   1:  PR[GP1:91,1] = PR[GP1:90,1] + -18.731;
   1:  PR[GP1:91,2] = PR[GP1:90,2] + 32.374;
   1:L PR[91] 10mm/sec CNT100;
   1:  PR[GP1:91,1] = PR[GP1:90,1] + -20.880;
   1:  PR[GP1:91,2] = PR[GP1:90,2] + 33.052;
   1:L PR[91] 10mm/sec CNT100;
   1:  PR[GP1:91,1] = PR[GP1:90,1] + -27.675;
   1:  PR[GP1:91,2] = PR[GP1:90,2] + 35.074;
   1:L PR[91] 10mm/sec CNT100;
   1:  PR[GP1:91,1] = PR[GP1:90,1] + -31.879;
   1:  PR[GP1:91,2] = PR[GP1:90,2] + 35.433;
   1:L PR[91] 10mm/sec CNT100;
   1:  PR[GP1:91,1] = PR[GP1:90,1] + -39.590;
   1:  PR[GP1:91,2] = PR[GP1:90,2] + 35.208;
   1:L PR[91] 10mm/sec CNT100;
   1:  PR[GP1:91,1] = PR[GP1:90,1] + -42.034;
   1:  PR[GP1:91,2] = PR[GP1:90,2] + 34.900;
   1:L PR[91] 10mm/sec CNT100;
   1:  PR[GP1:91,1] = PR[GP1:90,1] + -53.582;
   1:  PR[GP1:91,2] = PR[GP1:90,2] + 30.630;
   1:L PR[91] 10mm/sec CNT100;
   1:  PR[GP1:91,1] = PR[GP1:90,1] + -53.589;
   1:  PR[GP1:91,2] = PR[GP1:90,2] + 30.626;
   1:L PR[91] 10mm/sec CNT100;
   1:  PR[GP1:91,1] = PR[GP1:90,1] + -63.016;
   1:  PR[GP1:91,2] = PR[GP1:90,2] + 22.850;
   1:L PR[91] 10mm/sec CNT100;
   1:  PR[GP1:91,1] = PR[GP1:90,1] + -64.107;
   1:  PR[GP1:91,2] = PR[GP1:90,2] + 21.068;
   1:L PR[91] 10mm/sec CNT100;
   1:  PR[GP1:91,1] = PR[GP1:90,1] + -69.252;
   1:  PR[GP1:91,2] = PR[GP1:90,2] + 12.300;
   1:L PR[91] 10mm/sec CNT100;
   1:  PR[GP1:91,1] = PR[GP1:90,1] + -69.934;
   1:  PR[GP1:91,2] = PR[GP1:90,2] + 8.701;
   1:L PR[91] 10mm/sec CNT100;
   1:  PR[GP1:91,1] = PR[GP1:90,1] + -71.444;
   1:  PR[GP1:91,2] = PR[GP1:90,2] + 0.282;
   1:L PR[91] 10mm/sec CNT100;
   1:  PR[GP1:91,1] = PR[GP1:90,1] + -70.746;
   1:  PR[GP1:91,2] = PR[GP1:90,2] + -3.377;
   1:L PR[91] 10mm/sec CNT100;
   1:  PR[GP1:91,1] = PR[GP1:90,1] + -69.251;
   1:  PR[GP1:91,2] = PR[GP1:90,2] + -11.744;
   1:L PR[91] 10mm/sec CNT100;
   1:  PR[GP1:91,1] = PR[GP1:90,1] + -64.107;
   1:  PR[GP1:91,2] = PR[GP1:90,2] + -20.510;
   1:L PR[91] 10mm/sec CNT100;
   1:  PR[GP1:91,1] = PR[GP1:90,1] + -63.016;
   1:  PR[GP1:91,2] = PR[GP1:90,2] + -22.292;
   1:L PR[91] 10mm/sec CNT100;
   1:  PR[GP1:91,1] = PR[GP1:90,1] + -53.589;
   1:  PR[GP1:91,2] = PR[GP1:90,2] + -30.068;
   1:L PR[91] 10mm/sec CNT100;
   1:  PR[GP1:91,1] = PR[GP1:90,1] + -53.582;
   1:  PR[GP1:91,2] = PR[GP1:90,2] + -30.072;
   1:L PR[91] 10mm/sec CNT100;
   1:  PR[GP1:91,1] = PR[GP1:90,1] + -42.034;
   1:  PR[GP1:91,2] = PR[GP1:90,2] + -34.342;
   1:L PR[91] 10mm/sec CNT100;
   1:  PR[GP1:91,1] = PR[GP1:90,1] + -39.590;
   1:  PR[GP1:91,2] = PR[GP1:90,2] + -34.650;
   1:L PR[91] 10mm/sec CNT100;
   1:  PR[GP1:91,1] = PR[GP1:90,1] + -31.879;
   1:  PR[GP1:91,2] = PR[GP1:90,2] + -34.875;
   1:L PR[91] 10mm/sec CNT100;
   1:  PR[GP1:91,1] = PR[GP1:90,1] + -27.681;
   1:  PR[GP1:91,2] = PR[GP1:90,2] + -34.516;
   1:L PR[91] 10mm/sec CNT100;
   1:  PR[GP1:91,1] = PR[GP1:90,1] + -23.858;
   1:  PR[GP1:91,2] = PR[GP1:90,2] + -33.291;
   1:L PR[91] 10mm/sec CNT100;
   1:  PR[GP1:91,1] = PR[GP1:90,1] + -18.724;
   1:  PR[GP1:91,2] = PR[GP1:90,2] + -31.812;
   1:L PR[91] 10mm/sec CNT100;
   1:  PR[GP1:91,1] = PR[GP1:90,1] + -14.436;
   1:  PR[GP1:91,2] = PR[GP1:90,2] + -29.375;
   1:L PR[91] 10mm/sec CNT100;
   1:  PR[GP1:91,1] = PR[GP1:90,1] + -11.858;
   1:  PR[GP1:91,2] = PR[GP1:90,2] + -27.972;
   1:L PR[91] 10mm/sec CNT100;
   1:  PR[GP1:91,1] = PR[GP1:90,1] + -5.874;
   1:  PR[GP1:91,2] = PR[GP1:90,2] + -22.708;
   1:L PR[91] 10mm/sec CNT100;
   1:  PR[GP1:91,1] = PR[GP1:90,1] + -5.197;
   1:  PR[GP1:91,2] = PR[GP1:90,2] + -21.887;
   1:L PR[91] 10mm/sec CNT100;
   1:  PR[GP1:91,1] = PR[GP1:90,1] + -1.808;
   1:  PR[GP1:91,2] = PR[GP1:90,2] + -17.107;
   1:L PR[91] 10mm/sec CNT100;
   1:  PR[GP1:91,1] = PR[GP1:90,1] + 1.289;
   1:L PR[91] 10mm/sec CNT100;
   1:  PR[GP1:91,1] = PR[GP1:90,1] + 4.280;
   1:  PR[GP1:91,2] = PR[GP1:90,2] + -21.758;
   1:  PR[GP1:91,3] = PR[GP1:90,3] + 40.565;
   1:L PR[91] 10mm/sec CNT100;
   1:  PR[GP1:91,1] = PR[GP1:90,1] + 5.162;
   1:  PR[GP1:91,2] = PR[GP1:90,2] + -22.831;
   1:L PR[91] 10mm/sec CNT100;
   1:  PR[GP1:91,1] = PR[GP1:90,1] + 11.120;
   1:  PR[GP1:91,2] = PR[GP1:90,2] + -28.070;
   1:L PR[91] 10mm/sec CNT100;
   1:  PR[GP1:91,1] = PR[GP1:90,1] + 16.147;
   1:  PR[GP1:91,2] = PR[GP1:90,2] + -30.798;
   1:L PR[91] 10mm/sec CNT100;
   1:  PR[GP1:91,1] = PR[GP1:90,1] + 18.170;
   1:  PR[GP1:91,2] = PR[GP1:90,2] + -31.944;
   1:L PR[91] 10mm/sec CNT100;
   1:  PR[GP1:91,1] = PR[GP1:90,1] + 19.162;
   1:  PR[GP1:91,2] = PR[GP1:90,2] + -32.258;
   1:L PR[91] 10mm/sec CNT100;
   1:  PR[GP1:91,1] = PR[GP1:90,1] + 26.811;
   1:  PR[GP1:91,2] = PR[GP1:90,2] + -34.534;
   1:L PR[91] 10mm/sec CNT100;
   1:  PR[GP1:91,1] = PR[GP1:90,1] + 31.532;
   1:  PR[GP1:91,2] = PR[GP1:90,2] + -34.940;
   1:L PR[91] 10mm/sec CNT100;
   1:  PR[GP1:91,1] = PR[GP1:90,1] + 38.345;
   1:  PR[GP1:91,2] = PR[GP1:90,2] + -34.741;
   1:L PR[91] 10mm/sec CNT100;
   1:  PR[GP1:91,1] = PR[GP1:90,1] + 41.413;
   1:  PR[GP1:91,2] = PR[GP1:90,2] + -34.357;
   1:L PR[91] 10mm/sec CNT100;
   1:  PR[GP1:91,1] = PR[GP1:90,1] + 52.707;
   1:  PR[GP1:91,2] = PR[GP1:90,2] + -30.191;
   1:L PR[91] 10mm/sec CNT100;
   1:  PR[GP1:91,1] = PR[GP1:90,1] + 53.122;
   1:  PR[GP1:91,2] = PR[GP1:90,2] + -29.937;
   1:L PR[91] 10mm/sec CNT100;
   1:  PR[GP1:91,1] = PR[GP1:90,1] + 62.401;
   1:  PR[GP1:91,2] = PR[GP1:90,2] + -22.260;
   1:L PR[91] 10mm/sec CNT100;
   1:  PR[GP1:91,1] = PR[GP1:90,1] + 63.095;
   1:  PR[GP1:91,2] = PR[GP1:90,2] + -21.128;
   1:L PR[91] 10mm/sec CNT100;
   1:  PR[GP1:91,1] = PR[GP1:90,1] + 68.617;
   1:  PR[GP1:91,2] = PR[GP1:90,2] + -11.744;
   1:L PR[91] 10mm/sec CNT100;
   1:  PR[GP1:91,1] = PR[GP1:90,1] + 69.156;
   1:  PR[GP1:91,2] = PR[GP1:90,2] + -8.896;
   1:L PR[91] 10mm/sec CNT100;
   1:  PR[GP1:91,1] = PR[GP1:90,1] + 70.798;
   1:  PR[GP1:91,2] = PR[GP1:90,2] + 0.276;
   1:L PR[91] 10mm/sec CNT100;
   1:  PR[GP1:91,1] = PR[GP1:90,1] + 70.220;
   1:  PR[GP1:91,2] = PR[GP1:90,2] + 3.310;
   1:L PR[91] 10mm/sec CNT100;
   1:  PR[GP1:91,1] = PR[GP1:90,1] + 68.615;
   1:  PR[GP1:91,2] = PR[GP1:90,2] + 12.305;
   1:L PR[91] 10mm/sec CNT100;
   1:  PR[GP1:91,1] = PR[GP1:90,1] + 63.095;
   1:  PR[GP1:91,2] = PR[GP1:90,2] + 21.686;
   1:L PR[91] 10mm/sec CNT100;
   1:  PR[GP1:91,1] = PR[GP1:90,1] + 62.401;
   1:  PR[GP1:91,2] = PR[GP1:90,2] + 22.818;
   1:L PR[91] 10mm/sec CNT100;
   1:  PR[GP1:91,1] = PR[GP1:90,1] + 53.122;
   1:  PR[GP1:91,2] = PR[GP1:90,2] + 30.495;
   1:L PR[91] 10mm/sec CNT100;
   1:  PR[GP1:91,1] = PR[GP1:90,1] + 52.707;
   1:  PR[GP1:91,2] = PR[GP1:90,2] + 30.749;
   1:L PR[91] 10mm/sec CNT100;
   1:  PR[GP1:91,1] = PR[GP1:90,1] + 43.327;
   1:  PR[GP1:91,2] = PR[GP1:90,2] + 34.223;
   1:L PR[91] 10mm/sec CNT100;
   1:  PR[GP1:91,1] = PR[GP1:90,1] + 41.415;
   1:  PR[GP1:91,2] = PR[GP1:90,2] + 34.915;
   1:L PR[91] 10mm/sec CNT100;
   1:  PR[GP1:91,1] = PR[GP1:90,1] + 38.345;
   1:  PR[GP1:91,2] = PR[GP1:90,2] + 35.299;
   1:L PR[91] 10mm/sec CNT100;
   1:  PR[GP1:91,1] = PR[GP1:90,1] + 31.532;
   1:  PR[GP1:91,2] = PR[GP1:90,2] + 35.498;
   1:L PR[91] 10mm/sec CNT100;
   1:  PR[GP1:91,1] = PR[GP1:90,1] + 26.818;
   1:  PR[GP1:91,2] = PR[GP1:90,2] + 35.093;
   1:L PR[91] 10mm/sec CNT100;
   1:  PR[GP1:91,1] = PR[GP1:90,1] + 23.739;
   1:  PR[GP1:91,2] = PR[GP1:90,2] + 34.106;
   1:L PR[91] 10mm/sec CNT100;
   1:  PR[GP1:91,1] = PR[GP1:90,1] + 18.163;
   1:  PR[GP1:91,2] = PR[GP1:90,2] + 32.499;
   1:L PR[91] 10mm/sec CNT100;
   1:  PR[GP1:91,1] = PR[GP1:90,1] + 16.146;
   1:  PR[GP1:91,2] = PR[GP1:90,2] + 31.356;
   1:L PR[91] 10mm/sec CNT100;
   1:  PR[GP1:91,1] = PR[GP1:90,1] + 11.256;
   1:  PR[GP1:91,2] = PR[GP1:90,2] + 28.716;
   1:L PR[91] 10mm/sec CNT100;
   1:  PR[GP1:91,1] = PR[GP1:90,1] + 10.671;
   1:  PR[GP1:91,2] = PR[GP1:90,2] + 28.240;
   1:L PR[91] 10mm/sec CNT100;
   1:  PR[GP1:91,1] = PR[GP1:90,1] + 5.156;
   1:  PR[GP1:91,2] = PR[GP1:90,2] + 23.383;
   1:L PR[91] 10mm/sec CNT100;
   1:  PR[GP1:91,1] = PR[GP1:90,1] + 4.259;
   1:  PR[GP1:91,2] = PR[GP1:90,2] + 22.289;
   1:L PR[91] 10mm/sec CNT100;
   1:  PR[GP1:91,1] = PR[GP1:90,1] + 1.201;
   1:  PR[GP1:91,2] = PR[GP1:90,2] + 17.990;
   1:L PR[91] 10mm/sec CNT100;
   1:  PR[GP1:91,1] = PR[GP1:90,1] + -1.721;
   1:L PR[91] 10mm/sec CNT100;
   1:  PR[GP1:91,1] = PR[GP1:90,1] + -4.761;
   1:  PR[GP1:91,2] = PR[GP1:90,2] + 22.278;
   1:L PR[91] 10mm/sec CNT100;
   1:  PR[GP1:91,1] = PR[GP1:90,1] + -5.643;
   1:  PR[GP1:91,2] = PR[GP1:90,2] + 23.348;
   1:L PR[91] 10mm/sec CNT100;
   1:  PR[GP1:91,1] = PR[GP1:90,1] + -11.163;
   1:  PR[GP1:91,2] = PR[GP1:90,2] + 28.209;
   1:L PR[91] 10mm/sec CNT100;
   1:  PR[GP1:91,1] = PR[GP1:90,1] + -11.750;
   1:  PR[GP1:91,2] = PR[GP1:90,2] + 28.687;
   1:L PR[91] 10mm/sec CNT100;
   1:  PR[GP1:91,1] = PR[GP1:90,1] + -16.673;
   1:  PR[GP1:91,2] = PR[GP1:90,2] + 31.352;
   1:L PR[91] 10mm/sec CNT100;
   1:  PR[GP1:91,1] = PR[GP1:90,1] + -18.703;
   1:  PR[GP1:91,2] = PR[GP1:90,2] + 32.506;
   1:L PR[91] 10mm/sec CNT100;
   1:  PR[GP1:91,1] = PR[GP1:90,1] + -19.698;
   1:  PR[GP1:91,2] = PR[GP1:90,2] + 32.820;
   1:L PR[91] 10mm/sec CNT100;
   1:  PR[GP1:91,1] = PR[GP1:90,1] + -27.337;
   1:  PR[GP1:91,2] = PR[GP1:90,2] + 35.093;
   1:L PR[91] 10mm/sec CNT100;
   1:  PR[GP1:91,1] = PR[GP1:90,1] + -32.070;
   1:  PR[GP1:91,2] = PR[GP1:90,2] + 35.498;
   1:L PR[91] 10mm/sec CNT100;
   1:  PR[GP1:91,1] = PR[GP1:90,1] + -38.884;
   1:  PR[GP1:91,2] = PR[GP1:90,2] + 35.298;
   1:L PR[91] 10mm/sec CNT100;
   1:  PR[GP1:91,1] = PR[GP1:90,1] + -41.955;
   1:  PR[GP1:91,2] = PR[GP1:90,2] + 34.912;
   1:L PR[91] 10mm/sec CNT100;
   1:  PR[GP1:91,1] = PR[GP1:90,1] + -53.238;
   1:  PR[GP1:91,2] = PR[GP1:90,2] + 30.743;
   1:L PR[91] 10mm/sec CNT100;
   1:  PR[GP1:91,1] = PR[GP1:90,1] + -53.655;
   1:  PR[GP1:91,2] = PR[GP1:90,2] + 30.487;
   1:L PR[91] 10mm/sec CNT100;
   1:  PR[GP1:91,1] = PR[GP1:90,1] + -62.929;
   1:  PR[GP1:91,2] = PR[GP1:90,2] + 22.824;
   1:L PR[91] 10mm/sec CNT100;
   1:  PR[GP1:91,1] = PR[GP1:90,1] + -63.623;
   1:  PR[GP1:91,2] = PR[GP1:90,2] + 21.691;
   1:L PR[91] 10mm/sec CNT100;
   1:  PR[GP1:91,1] = PR[GP1:90,1] + -69.144;
   1:  PR[GP1:91,2] = PR[GP1:90,2] + 12.283;
   1:L PR[91] 10mm/sec CNT100;
   1:  PR[GP1:91,1] = PR[GP1:90,1] + -69.683;
   1:  PR[GP1:91,2] = PR[GP1:90,2] + 9.438;
   1:L PR[91] 10mm/sec CNT100;
   1:  PR[GP1:91,1] = PR[GP1:90,1] + -71.325;
   1:  PR[GP1:91,2] = PR[GP1:90,2] + 0.282;
   1:L PR[91] 10mm/sec CNT100;
   1:  PR[GP1:91,1] = PR[GP1:90,1] + -70.746;
   1:  PR[GP1:91,2] = PR[GP1:90,2] + -2.749;
   1:L PR[91] 10mm/sec CNT100;
   1:  PR[GP1:91,1] = PR[GP1:90,1] + -69.142;
   1:  PR[GP1:91,2] = PR[GP1:90,2] + -11.727;
   1:L PR[91] 10mm/sec CNT100;
   1:  PR[GP1:91,1] = PR[GP1:90,1] + -63.623;
   1:  PR[GP1:91,2] = PR[GP1:90,2] + -21.133;
   1:L PR[91] 10mm/sec CNT100;
   1:  PR[GP1:91,1] = PR[GP1:90,1] + -62.929;
   1:  PR[GP1:91,2] = PR[GP1:90,2] + -22.266;
   1:L PR[91] 10mm/sec CNT100;
   1:  PR[GP1:91,1] = PR[GP1:90,1] + -53.655;
   1:  PR[GP1:91,2] = PR[GP1:90,2] + -29.929;
   1:L PR[91] 10mm/sec CNT100;
   1:  PR[GP1:91,1] = PR[GP1:90,1] + -53.238;
   1:  PR[GP1:91,2] = PR[GP1:90,2] + -30.185;
   1:L PR[91] 10mm/sec CNT100;
   1:  PR[GP1:91,1] = PR[GP1:90,1] + -43.863;
   1:  PR[GP1:91,2] = PR[GP1:90,2] + -33.661;
   1:L PR[91] 10mm/sec CNT100;
   1:  PR[GP1:91,1] = PR[GP1:90,1] + -41.957;
   1:  PR[GP1:91,2] = PR[GP1:90,2] + -34.354;
   1:L PR[91] 10mm/sec CNT100;
   1:  PR[GP1:91,1] = PR[GP1:90,1] + -38.884;
   1:  PR[GP1:91,2] = PR[GP1:90,2] + -34.740;
   1:L PR[91] 10mm/sec CNT100;
   1:  PR[GP1:91,1] = PR[GP1:90,1] + -32.070;
   1:  PR[GP1:91,2] = PR[GP1:90,2] + -34.940;
   1:L PR[91] 10mm/sec CNT100;
   1:  PR[GP1:91,1] = PR[GP1:90,1] + -27.344;
   1:  PR[GP1:91,2] = PR[GP1:90,2] + -34.535;
   1:L PR[91] 10mm/sec CNT100;
   1:  PR[GP1:91,1] = PR[GP1:90,1] + -24.265;
   1:  PR[GP1:91,2] = PR[GP1:90,2] + -33.549;
   1:L PR[91] 10mm/sec CNT100;
   1:  PR[GP1:91,1] = PR[GP1:90,1] + -18.697;
   1:  PR[GP1:91,2] = PR[GP1:90,2] + -31.944;
   1:L PR[91] 10mm/sec CNT100;
   1:  PR[GP1:91,1] = PR[GP1:90,1] + -16.674;
   1:  PR[GP1:91,2] = PR[GP1:90,2] + -30.794;
   1:L PR[91] 10mm/sec CNT100;
   1:  PR[GP1:91,1] = PR[GP1:90,1] + -11.614;
   1:  PR[GP1:91,2] = PR[GP1:90,2] + -28.041;
   1:L PR[91] 10mm/sec CNT100;
   1:  PR[GP1:91,1] = PR[GP1:90,1] + -5.648;
   1:  PR[GP1:91,2] = PR[GP1:90,2] + -22.797;
   1:L PR[91] 10mm/sec CNT100;
   1:  PR[GP1:91,1] = PR[GP1:90,1] + -4.767;
   1:  PR[GP1:91,2] = PR[GP1:90,2] + -21.728;
   1:L PR[91] 10mm/sec CNT100;
   1:  PR[GP1:91,1] = PR[GP1:90,1] + -1.721;
   1:  PR[GP1:91,2] = PR[GP1:90,2] + -17.432;
   1:L PR[91] 10mm/sec CNT100;
   1:  PR[GP1:91,1] = PR[GP1:90,1] + 1.203;
   1:L PR[91] 10mm/sec CNT100;
   1:  PR[GP1:91,1] = PR[GP1:90,1] + 3.847;
   1:  PR[GP1:91,2] = PR[GP1:90,2] + -21.595;
   1:  PR[GP1:91,3] = PR[GP1:90,3] + 41.175;
   1:L PR[91] 10mm/sec CNT100;
   1:  PR[GP1:91,1] = PR[GP1:90,1] + 4.935;
   1:  PR[GP1:91,2] = PR[GP1:90,2] + -22.918;
   1:L PR[91] 10mm/sec CNT100;
   1:  PR[GP1:91,1] = PR[GP1:90,1] + 10.876;
   1:  PR[GP1:91,2] = PR[GP1:90,2] + -28.138;
   1:L PR[91] 10mm/sec CNT100;
   1:  PR[GP1:91,1] = PR[GP1:90,1] + 18.113;
   1:  PR[GP1:91,2] = PR[GP1:90,2] + -32.067;
   1:L PR[91] 10mm/sec CNT100;
   1:  PR[GP1:91,1] = PR[GP1:90,1] + 26.475;
   1:  PR[GP1:91,2] = PR[GP1:90,2] + -34.553;
   1:L PR[91] 10mm/sec CNT100;
   1:  PR[GP1:91,1] = PR[GP1:90,1] + 31.723;
   1:  PR[GP1:91,2] = PR[GP1:90,2] + -35.005;
   1:L PR[91] 10mm/sec CNT100;
   1:  PR[GP1:91,1] = PR[GP1:90,1] + 37.637;
   1:  PR[GP1:91,2] = PR[GP1:90,2] + -34.832;
   1:L PR[91] 10mm/sec CNT100;
   1:  PR[GP1:91,1] = PR[GP1:90,1] + 41.332;
   1:  PR[GP1:91,2] = PR[GP1:90,2] + -34.369;
   1:L PR[91] 10mm/sec CNT100;
   1:  PR[GP1:91,1] = PR[GP1:90,1] + 52.361;
   1:  PR[GP1:91,2] = PR[GP1:90,2] + -30.305;
   1:L PR[91] 10mm/sec CNT100;
   1:  PR[GP1:91,1] = PR[GP1:90,1] + 53.185;
   1:  PR[GP1:91,2] = PR[GP1:90,2] + -29.801;
   1:L PR[91] 10mm/sec CNT100;
   1:  PR[GP1:91,1] = PR[GP1:90,1] + 62.315;
   1:  PR[GP1:91,2] = PR[GP1:90,2] + -22.234;
   1:L PR[91] 10mm/sec CNT100;
   1:  PR[GP1:91,1] = PR[GP1:90,1] + 62.611;
   1:  PR[GP1:91,2] = PR[GP1:90,2] + -21.750;
   1:L PR[91] 10mm/sec CNT100;
   1:  PR[GP1:91,1] = PR[GP1:90,1] + 68.508;
   1:  PR[GP1:91,2] = PR[GP1:90,2] + -11.728;
   1:L PR[91] 10mm/sec CNT100;
   1:  PR[GP1:91,1] = PR[GP1:90,1] + 68.904;
   1:  PR[GP1:91,2] = PR[GP1:90,2] + -9.635;
   1:L PR[91] 10mm/sec CNT100;
   1:  PR[GP1:91,1] = PR[GP1:90,1] + 70.679;
   1:  PR[GP1:91,2] = PR[GP1:90,2] + 0.276;
   1:L PR[91] 10mm/sec CNT100;
   1:  PR[GP1:91,1] = PR[GP1:90,1] + 70.220;
   1:  PR[GP1:91,2] = PR[GP1:90,2] + 2.681;
   1:L PR[91] 10mm/sec CNT100;
   1:  PR[GP1:91,1] = PR[GP1:90,1] + 68.507;
   1:  PR[GP1:91,2] = PR[GP1:90,2] + 12.289;
   1:L PR[91] 10mm/sec CNT100;
   1:  PR[GP1:91,1] = PR[GP1:90,1] + 62.611;
   1:  PR[GP1:91,2] = PR[GP1:90,2] + 22.308;
   1:L PR[91] 10mm/sec CNT100;
   1:  PR[GP1:91,1] = PR[GP1:90,1] + 62.315;
   1:  PR[GP1:91,2] = PR[GP1:90,2] + 22.792;
   1:L PR[91] 10mm/sec CNT100;
   1:  PR[GP1:91,1] = PR[GP1:90,1] + 53.185;
   1:  PR[GP1:91,2] = PR[GP1:90,2] + 30.359;
   1:L PR[91] 10mm/sec CNT100;
   1:  PR[GP1:91,1] = PR[GP1:90,1] + 52.361;
   1:  PR[GP1:91,2] = PR[GP1:90,2] + 30.863;
   1:L PR[91] 10mm/sec CNT100;
   1:  PR[GP1:91,1] = PR[GP1:90,1] + 43.637;
   1:  PR[GP1:91,2] = PR[GP1:90,2] + 34.094;
   1:L PR[91] 10mm/sec CNT100;
   1:  PR[GP1:91,1] = PR[GP1:90,1] + 41.334;
   1:  PR[GP1:91,2] = PR[GP1:90,2] + 34.927;
   1:L PR[91] 10mm/sec CNT100;
   1:  PR[GP1:91,1] = PR[GP1:90,1] + 37.637;
   1:  PR[GP1:91,2] = PR[GP1:90,2] + 35.390;
   1:L PR[91] 10mm/sec CNT100;
   1:  PR[GP1:91,1] = PR[GP1:90,1] + 31.723;
   1:  PR[GP1:91,2] = PR[GP1:90,2] + 35.563;
   1:L PR[91] 10mm/sec CNT100;
   1:  PR[GP1:91,1] = PR[GP1:90,1] + 26.481;
   1:  PR[GP1:91,2] = PR[GP1:90,2] + 35.112;
   1:L PR[91] 10mm/sec CNT100;
   1:  PR[GP1:91,1] = PR[GP1:90,1] + 24.146;
   1:  PR[GP1:91,2] = PR[GP1:90,2] + 34.364;
   1:L PR[91] 10mm/sec CNT100;
   1:  PR[GP1:91,1] = PR[GP1:90,1] + 18.110;
   1:  PR[GP1:91,2] = PR[GP1:90,2] + 32.624;
   1:L PR[91] 10mm/sec CNT100;
   1:  PR[GP1:91,1] = PR[GP1:90,1] + 11.083;
   1:  PR[GP1:91,2] = PR[GP1:90,2] + 28.830;
   1:L PR[91] 10mm/sec CNT100;
   1:  PR[GP1:91,1] = PR[GP1:90,1] + 10.186;
   1:  PR[GP1:91,2] = PR[GP1:90,2] + 28.100;
   1:L PR[91] 10mm/sec CNT100;
   1:  PR[GP1:91,1] = PR[GP1:90,1] + 4.927;
   1:  PR[GP1:91,2] = PR[GP1:90,2] + 23.469;
   1:L PR[91] 10mm/sec CNT100;
   1:  PR[GP1:91,1] = PR[GP1:90,1] + 3.822;
   1:  PR[GP1:91,2] = PR[GP1:90,2] + 22.121;
   1:L PR[91] 10mm/sec CNT100;
   1:  PR[GP1:91,1] = PR[GP1:90,1] + 1.115;
   1:  PR[GP1:91,2] = PR[GP1:90,2] + 18.315;
   1:L PR[91] 10mm/sec CNT100;
   1:  PR[GP1:91,1] = PR[GP1:90,1] + -1.634;
   1:L PR[91] 10mm/sec CNT100;
   1:  PR[GP1:91,1] = PR[GP1:90,1] + -4.330;
   1:  PR[GP1:91,2] = PR[GP1:90,2] + 22.117;
   1:L PR[91] 10mm/sec CNT100;
   1:  PR[GP1:91,1] = PR[GP1:90,1] + -5.415;
   1:  PR[GP1:91,2] = PR[GP1:90,2] + 23.435;
   1:L PR[91] 10mm/sec CNT100;
   1:  PR[GP1:91,1] = PR[GP1:90,1] + -10.680;
   1:  PR[GP1:91,2] = PR[GP1:90,2] + 28.071;
   1:L PR[91] 10mm/sec CNT100;
   1:  PR[GP1:91,1] = PR[GP1:90,1] + -11.578;
   1:  PR[GP1:91,2] = PR[GP1:90,2] + 28.801;
   1:L PR[91] 10mm/sec CNT100;
   1:  PR[GP1:91,1] = PR[GP1:90,1] + -18.645;
   1:  PR[GP1:91,2] = PR[GP1:90,2] + 32.628;
   1:L PR[91] 10mm/sec CNT100;
   1:  PR[GP1:91,1] = PR[GP1:90,1] + -27.000;
   1:  PR[GP1:91,2] = PR[GP1:90,2] + 35.112;
   1:L PR[91] 10mm/sec CNT100;
   1:  PR[GP1:91,1] = PR[GP1:90,1] + -32.262;
   1:  PR[GP1:91,2] = PR[GP1:90,2] + 35.562;
   1:L PR[91] 10mm/sec CNT100;
   1:  PR[GP1:91,1] = PR[GP1:90,1] + -38.178;
   1:  PR[GP1:91,2] = PR[GP1:90,2] + 35.389;
   1:L PR[91] 10mm/sec CNT100;
   1:  PR[GP1:91,1] = PR[GP1:90,1] + -41.877;
   1:  PR[GP1:91,2] = PR[GP1:90,2] + 34.924;
   1:L PR[91] 10mm/sec CNT100;
   1:  PR[GP1:91,1] = PR[GP1:90,1] + -52.894;
   1:  PR[GP1:91,2] = PR[GP1:90,2] + 30.856;
   1:L PR[91] 10mm/sec CNT100;
   1:  PR[GP1:91,1] = PR[GP1:90,1] + -53.720;
   1:  PR[GP1:91,2] = PR[GP1:90,2] + 30.348;
   1:L PR[91] 10mm/sec CNT100;
   1:  PR[GP1:91,1] = PR[GP1:90,1] + -62.842;
   1:  PR[GP1:91,2] = PR[GP1:90,2] + 22.799;
   1:L PR[91] 10mm/sec CNT100;
   1:  PR[GP1:91,1] = PR[GP1:90,1] + -63.139;
   1:  PR[GP1:91,2] = PR[GP1:90,2] + 22.314;
   1:L PR[91] 10mm/sec CNT100;
   1:  PR[GP1:91,1] = PR[GP1:90,1] + -69.035;
   1:  PR[GP1:91,2] = PR[GP1:90,2] + 12.266;
   1:L PR[91] 10mm/sec CNT100;
   1:  PR[GP1:91,1] = PR[GP1:90,1] + -69.431;
   1:  PR[GP1:91,2] = PR[GP1:90,2] + 10.175;
   1:L PR[91] 10mm/sec CNT100;
   1:  PR[GP1:91,1] = PR[GP1:90,1] + -71.205;
   1:  PR[GP1:91,2] = PR[GP1:90,2] + 0.282;
   1:L PR[91] 10mm/sec CNT100;
   1:  PR[GP1:91,1] = PR[GP1:90,1] + -70.747;
   1:  PR[GP1:91,2] = PR[GP1:90,2] + -2.120;
   1:L PR[91] 10mm/sec CNT100;
   1:  PR[GP1:91,1] = PR[GP1:90,1] + -69.033;
   1:  PR[GP1:91,2] = PR[GP1:90,2] + -11.711;
   1:L PR[91] 10mm/sec CNT100;
   1:  PR[GP1:91,1] = PR[GP1:90,1] + -63.139;
   1:  PR[GP1:91,2] = PR[GP1:90,2] + -21.756;
   1:L PR[91] 10mm/sec CNT100;
   1:  PR[GP1:91,1] = PR[GP1:90,1] + -62.842;
   1:  PR[GP1:91,2] = PR[GP1:90,2] + -22.241;
   1:L PR[91] 10mm/sec CNT100;
   1:  PR[GP1:91,1] = PR[GP1:90,1] + -53.721;
   1:  PR[GP1:91,2] = PR[GP1:90,2] + -29.790;
   1:L PR[91] 10mm/sec CNT100;
   1:  PR[GP1:91,1] = PR[GP1:90,1] + -52.894;
   1:  PR[GP1:91,2] = PR[GP1:90,2] + -30.299;
   1:L PR[91] 10mm/sec CNT100;
   1:  PR[GP1:91,1] = PR[GP1:90,1] + -44.175;
   1:  PR[GP1:91,2] = PR[GP1:90,2] + -33.531;
   1:L PR[91] 10mm/sec CNT100;
   1:  PR[GP1:91,1] = PR[GP1:90,1] + -41.879;
   1:  PR[GP1:91,2] = PR[GP1:90,2] + -34.365;
   1:L PR[91] 10mm/sec CNT100;
   1:  PR[GP1:91,1] = PR[GP1:90,1] + -38.179;
   1:  PR[GP1:91,2] = PR[GP1:90,2] + -34.831;
   1:L PR[91] 10mm/sec CNT100;
   1:  PR[GP1:91,1] = PR[GP1:90,1] + -32.262;
   1:  PR[GP1:91,2] = PR[GP1:90,2] + -35.004;
   1:L PR[91] 10mm/sec CNT100;
   1:  PR[GP1:91,1] = PR[GP1:90,1] + -27.006;
   1:  PR[GP1:91,2] = PR[GP1:90,2] + -34.554;
   1:L PR[91] 10mm/sec CNT100;
   1:  PR[GP1:91,1] = PR[GP1:90,1] + -24.672;
   1:  PR[GP1:91,2] = PR[GP1:90,2] + -33.806;
   1:L PR[91] 10mm/sec CNT100;
   1:  PR[GP1:91,1] = PR[GP1:90,1] + -18.646;
   1:  PR[GP1:91,2] = PR[GP1:90,2] + -32.070;
   1:L PR[91] 10mm/sec CNT100;
   1:  PR[GP1:91,1] = PR[GP1:90,1] + -11.371;
   1:  PR[GP1:91,2] = PR[GP1:90,2] + -28.110;
   1:L PR[91] 10mm/sec CNT100;
   1:  PR[GP1:91,1] = PR[GP1:90,1] + -5.422;
   1:  PR[GP1:91,2] = PR[GP1:90,2] + -22.885;
   1:L PR[91] 10mm/sec CNT100;
   1:  PR[GP1:91,1] = PR[GP1:90,1] + -4.337;
   1:  PR[GP1:91,2] = PR[GP1:90,2] + -21.569;
   1:L PR[91] 10mm/sec CNT100;
   1:  PR[GP1:91,1] = PR[GP1:90,1] + -1.634;
   1:  PR[GP1:91,2] = PR[GP1:90,2] + -17.757;
   1:L PR[91] 10mm/sec CNT100;
   1:  PR[GP1:91,1] = PR[GP1:90,1] + 1.117;
   1:L PR[91] 10mm/sec CNT100;
   1:  PR[GP1:91,1] = PR[GP1:90,1] + 3.414;
   1:  PR[GP1:91,2] = PR[GP1:90,2] + -21.432;
   1:  PR[GP1:91,3] = PR[GP1:90,3] + 41.785;
   1:L PR[91] 10mm/sec CNT100;
   1:  PR[GP1:91,1] = PR[GP1:90,1] + 4.707;
   1:  PR[GP1:91,2] = PR[GP1:90,2] + -23.005;
   1:L PR[91] 10mm/sec CNT100;
   1:  PR[GP1:91,1] = PR[GP1:90,1] + 10.632;
   1:  PR[GP1:91,2] = PR[GP1:90,2] + -28.207;
   1:L PR[91] 10mm/sec CNT100;
   1:  PR[GP1:91,1] = PR[GP1:90,1] + 17.857;
   1:  PR[GP1:91,2] = PR[GP1:90,2] + -32.135;
   1:L PR[91] 10mm/sec CNT100;
   1:  PR[GP1:91,1] = PR[GP1:90,1] + 20.498;
   1:  PR[GP1:91,2] = PR[GP1:90,2] + -32.894;
   1:L PR[91] 10mm/sec CNT100;
   1:  PR[GP1:91,1] = PR[GP1:90,1] + 26.138;
   1:  PR[GP1:91,2] = PR[GP1:90,2] + -34.572;
   1:L PR[91] 10mm/sec CNT100;
   1:  PR[GP1:91,1] = PR[GP1:90,1] + 31.914;
   1:  PR[GP1:91,2] = PR[GP1:90,2] + -35.069;
   1:L PR[91] 10mm/sec CNT100;
   1:  PR[GP1:91,1] = PR[GP1:90,1] + 36.930;
   1:  PR[GP1:91,2] = PR[GP1:90,2] + -34.923;
   1:L PR[91] 10mm/sec CNT100;
   1:  PR[GP1:91,1] = PR[GP1:90,1] + 41.252;
   1:  PR[GP1:91,2] = PR[GP1:90,2] + -34.381;
   1:L PR[91] 10mm/sec CNT100;
   1:  PR[GP1:91,1] = PR[GP1:90,1] + 52.015;
   1:  PR[GP1:91,2] = PR[GP1:90,2] + -30.419;
   1:L PR[91] 10mm/sec CNT100;
   1:  PR[GP1:91,1] = PR[GP1:90,1] + 53.247;
   1:  PR[GP1:91,2] = PR[GP1:90,2] + -29.665;
   1:L PR[91] 10mm/sec CNT100;
   1:  PR[GP1:91,1] = PR[GP1:90,1] + 62.216;
   1:  PR[GP1:91,2] = PR[GP1:90,2] + -22.213;
   1:L PR[91] 10mm/sec CNT100;
   1:  PR[GP1:91,1] = PR[GP1:90,1] + 68.400;
   1:  PR[GP1:91,2] = PR[GP1:90,2] + -11.711;
   1:L PR[91] 10mm/sec CNT100;
   1:  PR[GP1:91,1] = PR[GP1:90,1] + 68.653;
   1:  PR[GP1:91,2] = PR[GP1:90,2] + -10.374;
   1:L PR[91] 10mm/sec CNT100;
   1:  PR[GP1:91,1] = PR[GP1:90,1] + 70.560;
   1:  PR[GP1:91,2] = PR[GP1:90,2] + 0.276;
   1:L PR[91] 10mm/sec CNT100;
   1:  PR[GP1:91,1] = PR[GP1:90,1] + 70.221;
   1:  PR[GP1:91,2] = PR[GP1:90,2] + 2.052;
   1:L PR[91] 10mm/sec CNT100;
   1:  PR[GP1:91,1] = PR[GP1:90,1] + 68.398;
   1:  PR[GP1:91,2] = PR[GP1:90,2] + 12.272;
   1:L PR[91] 10mm/sec CNT100;
   1:  PR[GP1:91,1] = PR[GP1:90,1] + 62.216;
   1:  PR[GP1:91,2] = PR[GP1:90,2] + 22.771;
   1:L PR[91] 10mm/sec CNT100;
   1:  PR[GP1:91,1] = PR[GP1:90,1] + 53.247;
   1:  PR[GP1:91,2] = PR[GP1:90,2] + 30.223;
   1:L PR[91] 10mm/sec CNT100;
   1:  PR[GP1:91,1] = PR[GP1:90,1] + 52.015;
   1:  PR[GP1:91,2] = PR[GP1:90,2] + 30.977;
   1:L PR[91] 10mm/sec CNT100;
   1:  PR[GP1:91,1] = PR[GP1:90,1] + 43.948;
   1:  PR[GP1:91,2] = PR[GP1:90,2] + 33.964;
   1:L PR[91] 10mm/sec CNT100;
   1:  PR[GP1:91,1] = PR[GP1:90,1] + 41.254;
   1:  PR[GP1:91,2] = PR[GP1:90,2] + 34.939;
   1:L PR[91] 10mm/sec CNT100;
   1:  PR[GP1:91,1] = PR[GP1:90,1] + 36.930;
   1:  PR[GP1:91,2] = PR[GP1:90,2] + 35.481;
   1:L PR[91] 10mm/sec CNT100;
   1:  PR[GP1:91,1] = PR[GP1:90,1] + 31.914;
   1:  PR[GP1:91,2] = PR[GP1:90,2] + 35.627;
   1:L PR[91] 10mm/sec CNT100;
   1:  PR[GP1:91,1] = PR[GP1:90,1] + 26.144;
   1:  PR[GP1:91,2] = PR[GP1:90,2] + 35.131;
   1:L PR[91] 10mm/sec CNT100;
   1:  PR[GP1:91,1] = PR[GP1:90,1] + 24.554;
   1:  PR[GP1:91,2] = PR[GP1:90,2] + 34.621;
   1:L PR[91] 10mm/sec CNT100;
   1:  PR[GP1:91,1] = PR[GP1:90,1] + 17.852;
   1:  PR[GP1:91,2] = PR[GP1:90,2] + 32.691;
   1:L PR[91] 10mm/sec CNT100;
   1:  PR[GP1:91,1] = PR[GP1:90,1] + 10.910;
   1:  PR[GP1:91,2] = PR[GP1:90,2] + 28.944;
   1:L PR[91] 10mm/sec CNT100;
   1:  PR[GP1:91,1] = PR[GP1:90,1] + 9.702;
   1:  PR[GP1:91,2] = PR[GP1:90,2] + 27.961;
   1:L PR[91] 10mm/sec CNT100;
   1:  PR[GP1:91,1] = PR[GP1:90,1] + 4.698;
   1:  PR[GP1:91,2] = PR[GP1:90,2] + 23.554;
   1:L PR[91] 10mm/sec CNT100;
   1:  PR[GP1:91,1] = PR[GP1:90,1] + 3.384;
   1:  PR[GP1:91,2] = PR[GP1:90,2] + 21.952;
   1:L PR[91] 10mm/sec CNT100;
   1:  PR[GP1:91,1] = PR[GP1:90,1] + 1.028;
   1:  PR[GP1:91,2] = PR[GP1:90,2] + 18.640;
   1:L PR[91] 10mm/sec CNT100;
   1:  PR[GP1:91,1] = PR[GP1:90,1] + -1.547;
   1:L PR[91] 10mm/sec CNT100;
   1:  PR[GP1:91,1] = PR[GP1:90,1] + -3.898;
   1:  PR[GP1:91,2] = PR[GP1:90,2] + 21.956;
   1:L PR[91] 10mm/sec CNT100;
   1:  PR[GP1:91,1] = PR[GP1:90,1] + -5.188;
   1:  PR[GP1:91,2] = PR[GP1:90,2] + 23.523;
   1:L PR[91] 10mm/sec CNT100;
   1:  PR[GP1:91,1] = PR[GP1:90,1] + -10.196;
   1:  PR[GP1:91,2] = PR[GP1:90,2] + 27.933;
   1:L PR[91] 10mm/sec CNT100;
   1:  PR[GP1:91,1] = PR[GP1:90,1] + -11.406;
   1:  PR[GP1:91,2] = PR[GP1:90,2] + 28.916;
   1:L PR[91] 10mm/sec CNT100;
   1:  PR[GP1:91,1] = PR[GP1:90,1] + -18.386;
   1:  PR[GP1:91,2] = PR[GP1:90,2] + 32.695;
   1:L PR[91] 10mm/sec CNT100;
   1:  PR[GP1:91,1] = PR[GP1:90,1] + -21.025;
   1:  PR[GP1:91,2] = PR[GP1:90,2] + 33.454;
   1:L PR[91] 10mm/sec CNT100;
   1:  PR[GP1:91,1] = PR[GP1:90,1] + -26.663;
   1:  PR[GP1:91,2] = PR[GP1:90,2] + 35.131;
   1:L PR[91] 10mm/sec CNT100;
   1:  PR[GP1:91,1] = PR[GP1:90,1] + -32.454;
   1:  PR[GP1:91,2] = PR[GP1:90,2] + 35.627;
   1:L PR[91] 10mm/sec CNT100;
   1:  PR[GP1:91,1] = PR[GP1:90,1] + -37.473;
   1:  PR[GP1:91,2] = PR[GP1:90,2] + 35.480;
   1:L PR[91] 10mm/sec CNT100;
   1:  PR[GP1:91,1] = PR[GP1:90,1] + -41.799;
   1:  PR[GP1:91,2] = PR[GP1:90,2] + 34.935;
   1:L PR[91] 10mm/sec CNT100;
   1:  PR[GP1:91,1] = PR[GP1:90,1] + -52.550;
   1:  PR[GP1:91,2] = PR[GP1:90,2] + 30.970;
   1:L PR[91] 10mm/sec CNT100;
   1:  PR[GP1:91,1] = PR[GP1:90,1] + -53.786;
   1:  PR[GP1:91,2] = PR[GP1:90,2] + 30.209;
   1:L PR[91] 10mm/sec CNT100;
   1:  PR[GP1:91,1] = PR[GP1:90,1] + -62.738;
   1:  PR[GP1:91,2] = PR[GP1:90,2] + 22.789;
   1:L PR[91] 10mm/sec CNT100;
   1:  PR[GP1:91,1] = PR[GP1:90,1] + -63.052;
   1:  PR[GP1:91,2] = PR[GP1:90,2] + 22.260;
   1:L PR[91] 10mm/sec CNT100;
   1:  PR[GP1:91,1] = PR[GP1:90,1] + -68.926;
   1:  PR[GP1:91,2] = PR[GP1:90,2] + 12.249;
   1:L PR[91] 10mm/sec CNT100;
   1:  PR[GP1:91,1] = PR[GP1:90,1] + -69.180;
   1:  PR[GP1:91,2] = PR[GP1:90,2] + 10.912;
   1:L PR[91] 10mm/sec CNT100;
   1:  PR[GP1:91,1] = PR[GP1:90,1] + -71.086;
   1:  PR[GP1:91,2] = PR[GP1:90,2] + 0.282;
   1:L PR[91] 10mm/sec CNT100;
   1:  PR[GP1:91,1] = PR[GP1:90,1] + -70.748;
   1:  PR[GP1:91,2] = PR[GP1:90,2] + -1.492;
   1:L PR[91] 10mm/sec CNT100;
   1:  PR[GP1:91,1] = PR[GP1:90,1] + -68.925;
   1:  PR[GP1:91,2] = PR[GP1:90,2] + -11.694;
   1:L PR[91] 10mm/sec CNT100;
   1:  PR[GP1:91,1] = PR[GP1:90,1] + -63.052;
   1:  PR[GP1:91,2] = PR[GP1:90,2] + -21.702;
   1:L PR[91] 10mm/sec CNT100;
   1:  PR[GP1:91,1] = PR[GP1:90,1] + -62.742;
   1:  PR[GP1:91,2] = PR[GP1:90,2] + -22.227;
   1:L PR[91] 10mm/sec CNT100;
   1:  PR[GP1:91,1] = PR[GP1:90,1] + -62.740;
   1:  PR[GP1:91,2] = PR[GP1:90,2] + -22.229;
   1:L PR[91] 10mm/sec CNT100;
   1:  PR[GP1:91,1] = PR[GP1:90,1] + -53.786;
   1:  PR[GP1:91,2] = PR[GP1:90,2] + -29.651;
   1:L PR[91] 10mm/sec CNT100;
   1:  PR[GP1:91,1] = PR[GP1:90,1] + -52.550;
   1:  PR[GP1:91,2] = PR[GP1:90,2] + -30.412;
   1:L PR[91] 10mm/sec CNT100;
   1:  PR[GP1:91,1] = PR[GP1:90,1] + -44.487;
   1:  PR[GP1:91,2] = PR[GP1:90,2] + -33.401;
   1:L PR[91] 10mm/sec CNT100;
   1:  PR[GP1:91,1] = PR[GP1:90,1] + -41.800;
   1:  PR[GP1:91,2] = PR[GP1:90,2] + -34.377;
   1:L PR[91] 10mm/sec CNT100;
   1:  PR[GP1:91,1] = PR[GP1:90,1] + -37.473;
   1:  PR[GP1:91,2] = PR[GP1:90,2] + -34.922;
   1:L PR[91] 10mm/sec CNT100;
   1:  PR[GP1:91,1] = PR[GP1:90,1] + -32.454;
   1:  PR[GP1:91,2] = PR[GP1:90,2] + -35.069;
   1:L PR[91] 10mm/sec CNT100;
   1:  PR[GP1:91,1] = PR[GP1:90,1] + -26.669;
   1:  PR[GP1:91,2] = PR[GP1:90,2] + -34.573;
   1:L PR[91] 10mm/sec CNT100;
   1:  PR[GP1:91,1] = PR[GP1:90,1] + -25.079;
   1:  PR[GP1:91,2] = PR[GP1:90,2] + -34.064;
   1:L PR[91] 10mm/sec CNT100;
   1:  PR[GP1:91,1] = PR[GP1:90,1] + -18.391;
   1:  PR[GP1:91,2] = PR[GP1:90,2] + -32.139;
   1:L PR[91] 10mm/sec CNT100;
   1:  PR[GP1:91,1] = PR[GP1:90,1] + -11.125;
   1:  PR[GP1:91,2] = PR[GP1:90,2] + -28.178;
   1:L PR[91] 10mm/sec CNT100;
   1:  PR[GP1:91,1] = PR[GP1:90,1] + -10.216;
   1:  PR[GP1:91,2] = PR[GP1:90,2] + -27.393;
   1:L PR[91] 10mm/sec CNT100;
   1:  PR[GP1:91,1] = PR[GP1:90,1] + -5.196;
   1:  PR[GP1:91,2] = PR[GP1:90,2] + -22.974;
   1:L PR[91] 10mm/sec CNT100;
   1:  PR[GP1:91,1] = PR[GP1:90,1] + -3.907;
   1:  PR[GP1:91,2] = PR[GP1:90,2] + -21.409;
   1:L PR[91] 10mm/sec CNT100;
   1:  PR[GP1:91,1] = PR[GP1:90,1] + -1.547;
   1:  PR[GP1:91,2] = PR[GP1:90,2] + -18.082;
   1:L PR[91] 10mm/sec CNT100;
   1:  PR[GP1:91,1] = PR[GP1:90,1] + 1.031;
   1:L PR[91] 10mm/sec CNT100;
   1:  PR[GP1:91,1] = PR[GP1:90,1] + 2.980;
   1:  PR[GP1:91,2] = PR[GP1:90,2] + -21.269;
   1:  PR[GP1:91,3] = PR[GP1:90,3] + 42.395;
   1:L PR[91] 10mm/sec CNT100;
   1:  PR[GP1:91,1] = PR[GP1:90,1] + 4.480;
   1:  PR[GP1:91,2] = PR[GP1:90,2] + -23.092;
   1:L PR[91] 10mm/sec CNT100;
   1:  PR[GP1:91,1] = PR[GP1:90,1] + 9.240;
   1:  PR[GP1:91,2] = PR[GP1:90,2] + -27.284;
   1:L PR[91] 10mm/sec CNT100;
   1:  PR[GP1:91,1] = PR[GP1:90,1] + 10.385;
   1:  PR[GP1:91,2] = PR[GP1:90,2] + -28.274;
   1:L PR[91] 10mm/sec CNT100;
   1:  PR[GP1:91,1] = PR[GP1:90,1] + 17.343;
   1:  PR[GP1:91,2] = PR[GP1:90,2] + -32.050;
   1:L PR[91] 10mm/sec CNT100;
   1:  PR[GP1:91,1] = PR[GP1:90,1] + 17.611;
   1:  PR[GP1:91,2] = PR[GP1:90,2] + -32.207;
   1:L PR[91] 10mm/sec CNT100;
   1:  PR[GP1:91,1] = PR[GP1:90,1] + 22.736;
   1:  PR[GP1:91,2] = PR[GP1:90,2] + -33.679;
   1:L PR[91] 10mm/sec CNT100;
   1:  PR[GP1:91,1] = PR[GP1:90,1] + 25.801;
   1:  PR[GP1:91,2] = PR[GP1:90,2] + -34.591;
   1:L PR[91] 10mm/sec CNT100;
   1:  PR[GP1:91,1] = PR[GP1:90,1] + 32.105;
   1:  PR[GP1:91,2] = PR[GP1:90,2] + -35.134;
   1:L PR[91] 10mm/sec CNT100;
   1:  PR[GP1:91,1] = PR[GP1:90,1] + 36.222;
   1:  PR[GP1:91,2] = PR[GP1:90,2] + -35.014;
   1:L PR[91] 10mm/sec CNT100;
   1:  PR[GP1:91,1] = PR[GP1:90,1] + 41.171;
   1:  PR[GP1:91,2] = PR[GP1:90,2] + -34.393;
   1:L PR[91] 10mm/sec CNT100;
   1:  PR[GP1:91,1] = PR[GP1:90,1] + 48.818;
   1:  PR[GP1:91,2] = PR[GP1:90,2] + -31.570;
   1:L PR[91] 10mm/sec CNT100;
   1:  PR[GP1:91,1] = PR[GP1:90,1] + 51.670;
   1:  PR[GP1:91,2] = PR[GP1:90,2] + -30.532;
   1:L PR[91] 10mm/sec CNT100;
   1:  PR[GP1:91,1] = PR[GP1:90,1] + 53.310;
   1:  PR[GP1:91,2] = PR[GP1:90,2] + -29.529;
   1:L PR[91] 10mm/sec CNT100;
   1:  PR[GP1:91,1] = PR[GP1:90,1] + 61.707;
   1:  PR[GP1:91,2] = PR[GP1:90,2] + -22.557;
   1:L PR[91] 10mm/sec CNT100;
   1:  PR[GP1:91,1] = PR[GP1:90,1] + 62.053;
   1:  PR[GP1:91,2] = PR[GP1:90,2] + -22.221;
   1:L PR[91] 10mm/sec CNT100;
   1:  PR[GP1:91,1] = PR[GP1:90,1] + 65.517;
   1:  PR[GP1:91,2] = PR[GP1:90,2] + -16.410;
   1:L PR[91] 10mm/sec CNT100;
   1:  PR[GP1:91,1] = PR[GP1:90,1] + 68.290;
   1:  PR[GP1:91,2] = PR[GP1:90,2] + -11.698;
   1:L PR[91] 10mm/sec CNT100;
   1:  PR[GP1:91,1] = PR[GP1:90,1] + 70.441;
   1:  PR[GP1:91,2] = PR[GP1:90,2] + 0.276;
   1:L PR[91] 10mm/sec CNT100;
   1:  PR[GP1:91,1] = PR[GP1:90,1] + 70.222;
   1:  PR[GP1:91,2] = PR[GP1:90,2] + 1.423;
   1:L PR[91] 10mm/sec CNT100;
   1:  PR[GP1:91,1] = PR[GP1:90,1] + 68.290;
   1:  PR[GP1:91,2] = PR[GP1:90,2] + 12.255;
   1:L PR[91] 10mm/sec CNT100;
   1:  PR[GP1:91,1] = PR[GP1:90,1] + 62.272;
   1:  PR[GP1:91,2] = PR[GP1:90,2] + 22.444;
   1:L PR[91] 10mm/sec CNT100;
   1:  PR[GP1:91,1] = PR[GP1:90,1] + 62.061;
   1:  PR[GP1:91,2] = PR[GP1:90,2] + 22.772;
   1:L PR[91] 10mm/sec CNT100;
   1:  PR[GP1:91,1] = PR[GP1:90,1] + 61.707;
   1:  PR[GP1:91,2] = PR[GP1:90,2] + 23.115;
   1:L PR[91] 10mm/sec CNT100;
   1:  PR[GP1:91,1] = PR[GP1:90,1] + 53.310;
   1:  PR[GP1:91,2] = PR[GP1:90,2] + 30.087;
   1:L PR[91] 10mm/sec CNT100;
   1:  PR[GP1:91,1] = PR[GP1:90,1] + 51.669;
   1:  PR[GP1:91,2] = PR[GP1:90,2] + 31.091;
   1:L PR[91] 10mm/sec CNT100;
   1:  PR[GP1:91,1] = PR[GP1:90,1] + 44.259;
   1:  PR[GP1:91,2] = PR[GP1:90,2] + 33.835;
   1:L PR[91] 10mm/sec CNT100;
   1:  PR[GP1:91,1] = PR[GP1:90,1] + 41.173;
   1:  PR[GP1:91,2] = PR[GP1:90,2] + 34.951;
   1:L PR[91] 10mm/sec CNT100;
   1:  PR[GP1:91,1] = PR[GP1:90,1] + 36.222;
   1:  PR[GP1:91,2] = PR[GP1:90,2] + 35.572;
   1:L PR[91] 10mm/sec CNT100;
   1:  PR[GP1:91,1] = PR[GP1:90,1] + 32.105;
   1:  PR[GP1:91,2] = PR[GP1:90,2] + 35.692;
   1:L PR[91] 10mm/sec CNT100;
   1:  PR[GP1:91,1] = PR[GP1:90,1] + 25.808;
   1:  PR[GP1:91,2] = PR[GP1:90,2] + 35.150;
   1:L PR[91] 10mm/sec CNT100;
   1:  PR[GP1:91,1] = PR[GP1:90,1] + 24.961;
   1:  PR[GP1:91,2] = PR[GP1:90,2] + 34.879;
   1:L PR[91] 10mm/sec CNT100;
   1:  PR[GP1:91,1] = PR[GP1:90,1] + 17.594;
   1:  PR[GP1:91,2] = PR[GP1:90,2] + 32.759;
   1:L PR[91] 10mm/sec CNT100;
   1:  PR[GP1:91,1] = PR[GP1:90,1] + 10.738;
   1:  PR[GP1:91,2] = PR[GP1:90,2] + 29.058;
   1:L PR[91] 10mm/sec CNT100;
   1:  PR[GP1:91,1] = PR[GP1:90,1] + 9.217;
   1:  PR[GP1:91,2] = PR[GP1:90,2] + 27.821;
   1:L PR[91] 10mm/sec CNT100;
   1:  PR[GP1:91,1] = PR[GP1:90,1] + 4.469;
   1:  PR[GP1:91,2] = PR[GP1:90,2] + 23.640;
   1:L PR[91] 10mm/sec CNT100;
   1:  PR[GP1:91,1] = PR[GP1:90,1] + 2.947;
   1:  PR[GP1:91,2] = PR[GP1:90,2] + 21.783;
   1:L PR[91] 10mm/sec CNT100;
   1:  PR[GP1:91,1] = PR[GP1:90,1] + 0.942;
   1:  PR[GP1:91,2] = PR[GP1:90,2] + 18.965;
   1:L PR[91] 10mm/sec CNT100;
   1:  PR[GP1:91,1] = PR[GP1:90,1] + -1.460;
   1:L PR[91] 10mm/sec CNT100;
   1:  PR[GP1:91,1] = PR[GP1:90,1] + -3.467;
   1:  PR[GP1:91,2] = PR[GP1:90,2] + 21.795;
   1:L PR[91] 10mm/sec CNT100;
   1:  PR[GP1:91,1] = PR[GP1:90,1] + -4.960;
   1:  PR[GP1:91,2] = PR[GP1:90,2] + 23.610;
   1:L PR[91] 10mm/sec CNT100;
   1:  PR[GP1:91,1] = PR[GP1:90,1] + -9.713;
   1:  PR[GP1:91,2] = PR[GP1:90,2] + 27.794;
   1:L PR[91] 10mm/sec CNT100;
   1:  PR[GP1:91,1] = PR[GP1:90,1] + -11.233;
   1:  PR[GP1:91,2] = PR[GP1:90,2] + 29.030;
   1:L PR[91] 10mm/sec CNT100;
   1:  PR[GP1:91,1] = PR[GP1:90,1] + -18.128;
   1:  PR[GP1:91,2] = PR[GP1:90,2] + 32.763;
   1:L PR[91] 10mm/sec CNT100;
   1:  PR[GP1:91,1] = PR[GP1:90,1] + -23.262;
   1:  PR[GP1:91,2] = PR[GP1:90,2] + 34.239;
   1:L PR[91] 10mm/sec CNT100;
   1:  PR[GP1:91,1] = PR[GP1:90,1] + -26.325;
   1:  PR[GP1:91,2] = PR[GP1:90,2] + 35.150;
   1:L PR[91] 10mm/sec CNT100;
   1:  PR[GP1:91,1] = PR[GP1:90,1] + -32.646;
   1:  PR[GP1:91,2] = PR[GP1:90,2] + 35.691;
   1:L PR[91] 10mm/sec CNT100;
   1:  PR[GP1:91,1] = PR[GP1:90,1] + -36.767;
   1:  PR[GP1:91,2] = PR[GP1:90,2] + 35.570;
   1:L PR[91] 10mm/sec CNT100;
   1:  PR[GP1:91,1] = PR[GP1:90,1] + -41.721;
   1:  PR[GP1:91,2] = PR[GP1:90,2] + 34.947;
   1:L PR[91] 10mm/sec CNT100;
   1:  PR[GP1:91,1] = PR[GP1:90,1] + -52.206;
   1:  PR[GP1:91,2] = PR[GP1:90,2] + 31.083;
   1:L PR[91] 10mm/sec CNT100;
   1:  PR[GP1:91,1] = PR[GP1:90,1] + -53.852;
   1:  PR[GP1:91,2] = PR[GP1:90,2] + 30.070;
   1:L PR[91] 10mm/sec CNT100;
   1:  PR[GP1:91,1] = PR[GP1:90,1] + -62.241;
   1:  PR[GP1:91,2] = PR[GP1:90,2] + 23.117;
   1:L PR[91] 10mm/sec CNT100;
   1:  PR[GP1:91,1] = PR[GP1:90,1] + -62.585;
   1:  PR[GP1:91,2] = PR[GP1:90,2] + 22.782;
   1:L PR[91] 10mm/sec CNT100;
   1:  PR[GP1:91,1] = PR[GP1:90,1] + -66.044;
   1:  PR[GP1:91,2] = PR[GP1:90,2] + 16.960;
   1:L PR[91] 10mm/sec CNT100;
   1:  PR[GP1:91,1] = PR[GP1:90,1] + -68.816;
   1:  PR[GP1:91,2] = PR[GP1:90,2] + 12.235;
   1:L PR[91] 10mm/sec CNT100;
   1:  PR[GP1:91,1] = PR[GP1:90,1] + -70.967;
   1:  PR[GP1:91,2] = PR[GP1:90,2] + 0.282;
   1:L PR[91] 10mm/sec CNT100;
   1:  PR[GP1:91,1] = PR[GP1:90,1] + -70.748;
   1:  PR[GP1:91,2] = PR[GP1:90,2] + -0.863;
   1:L PR[91] 10mm/sec CNT100;
   1:  PR[GP1:91,1] = PR[GP1:90,1] + -68.816;
   1:  PR[GP1:91,2] = PR[GP1:90,2] + -11.676;
   1:L PR[91] 10mm/sec CNT100;
   1:  PR[GP1:91,1] = PR[GP1:90,1] + -62.800;
   1:  PR[GP1:91,2] = PR[GP1:90,2] + -21.892;
   1:L PR[91] 10mm/sec CNT100;
   1:  PR[GP1:91,1] = PR[GP1:90,1] + -62.592;
   1:  PR[GP1:91,2] = PR[GP1:90,2] + -22.217;
   1:L PR[91] 10mm/sec CNT100;
   1:  PR[GP1:91,1] = PR[GP1:90,1] + -62.241;
   1:  PR[GP1:91,2] = PR[GP1:90,2] + -22.559;
   1:L PR[91] 10mm/sec CNT100;
   1:  PR[GP1:91,1] = PR[GP1:90,1] + -53.852;
   1:  PR[GP1:91,2] = PR[GP1:90,2] + -29.512;
   1:L PR[91] 10mm/sec CNT100;
   1:  PR[GP1:91,1] = PR[GP1:90,1] + -52.205;
   1:  PR[GP1:91,2] = PR[GP1:90,2] + -30.525;
   1:L PR[91] 10mm/sec CNT100;
   1:  PR[GP1:91,1] = PR[GP1:90,1] + -44.799;
   1:  PR[GP1:91,2] = PR[GP1:90,2] + -33.271;
   1:L PR[91] 10mm/sec CNT100;
   1:  PR[GP1:91,1] = PR[GP1:90,1] + -41.722;
   1:  PR[GP1:91,2] = PR[GP1:90,2] + -34.389;
   1:L PR[91] 10mm/sec CNT100;
   1:  PR[GP1:91,1] = PR[GP1:90,1] + -36.767;
   1:  PR[GP1:91,2] = PR[GP1:90,2] + -35.012;
   1:L PR[91] 10mm/sec CNT100;
   1:  PR[GP1:91,1] = PR[GP1:90,1] + -32.646;
   1:  PR[GP1:91,2] = PR[GP1:90,2] + -35.133;
   1:L PR[91] 10mm/sec CNT100;
   1:  PR[GP1:91,1] = PR[GP1:90,1] + -26.332;
   1:  PR[GP1:91,2] = PR[GP1:90,2] + -34.593;
   1:L PR[91] 10mm/sec CNT100;
   1:  PR[GP1:91,1] = PR[GP1:90,1] + -25.485;
   1:  PR[GP1:91,2] = PR[GP1:90,2] + -34.321;
   1:L PR[91] 10mm/sec CNT100;
   1:  PR[GP1:91,1] = PR[GP1:90,1] + -18.145;
   1:  PR[GP1:91,2] = PR[GP1:90,2] + -32.211;
   1:L PR[91] 10mm/sec CNT100;
   1:  PR[GP1:91,1] = PR[GP1:90,1] + -17.878;
   1:  PR[GP1:91,2] = PR[GP1:90,2] + -32.054;
   1:L PR[91] 10mm/sec CNT100;
   1:  PR[GP1:91,1] = PR[GP1:90,1] + -10.881;
   1:  PR[GP1:91,2] = PR[GP1:90,2] + -28.246;
   1:L PR[91] 10mm/sec CNT100;
   1:  PR[GP1:91,1] = PR[GP1:90,1] + -9.736;
   1:  PR[GP1:91,2] = PR[GP1:90,2] + -27.258;
   1:L PR[91] 10mm/sec CNT100;
   1:  PR[GP1:91,1] = PR[GP1:90,1] + -4.970;
   1:  PR[GP1:91,2] = PR[GP1:90,2] + -23.062;
   1:L PR[91] 10mm/sec CNT100;
   1:  PR[GP1:91,1] = PR[GP1:90,1] + -3.477;
   1:  PR[GP1:91,2] = PR[GP1:90,2] + -21.250;
   1:L PR[91] 10mm/sec CNT100;
   1:  PR[GP1:91,1] = PR[GP1:90,1] + -1.461;
   1:  PR[GP1:91,2] = PR[GP1:90,2] + -18.407;
   1:L PR[91] 10mm/sec CNT100;
   1:  PR[GP1:91,1] = PR[GP1:90,1] + 0.945;
   1:L PR[91] 10mm/sec CNT100;
   1:  PR[GP1:91,1] = PR[GP1:90,1] + 2.547;
   1:  PR[GP1:91,2] = PR[GP1:90,2] + -21.106;
   1:  PR[GP1:91,3] = PR[GP1:90,3] + 43.005;
   1:L PR[91] 10mm/sec CNT100;
   1:  PR[GP1:91,1] = PR[GP1:90,1] + 4.252;
   1:  PR[GP1:91,2] = PR[GP1:90,2] + -23.179;
   1:L PR[91] 10mm/sec CNT100;
   1:  PR[GP1:91,1] = PR[GP1:90,1] + 8.759;
   1:  PR[GP1:91,2] = PR[GP1:90,2] + -27.148;
   1:L PR[91] 10mm/sec CNT100;
   1:  PR[GP1:91,1] = PR[GP1:90,1] + 10.140;
   1:  PR[GP1:91,2] = PR[GP1:90,2] + -28.342;
   1:L PR[91] 10mm/sec CNT100;
   1:  PR[GP1:91,1] = PR[GP1:90,1] + 16.932;
   1:  PR[GP1:91,2] = PR[GP1:90,2] + -32.028;
   1:L PR[91] 10mm/sec CNT100;
   1:  PR[GP1:91,1] = PR[GP1:90,1] + 17.357;
   1:  PR[GP1:91,2] = PR[GP1:90,2] + -32.277;
   1:L PR[91] 10mm/sec CNT100;
   1:  PR[GP1:91,1] = PR[GP1:90,1] + 25.462;
   1:  PR[GP1:91,2] = PR[GP1:90,2] + -34.610;
   1:L PR[91] 10mm/sec CNT100;
   1:  PR[GP1:91,1] = PR[GP1:90,1] + 32.296;
   1:  PR[GP1:91,2] = PR[GP1:90,2] + -35.198;
   1:L PR[91] 10mm/sec CNT100;
   1:  PR[GP1:91,1] = PR[GP1:90,1] + 35.515;
   1:  PR[GP1:91,2] = PR[GP1:90,2] + -35.104;
   1:L PR[91] 10mm/sec CNT100;
   1:  PR[GP1:91,1] = PR[GP1:90,1] + 41.090;
   1:  PR[GP1:91,2] = PR[GP1:90,2] + -34.406;
   1:L PR[91] 10mm/sec CNT100;
   1:  PR[GP1:91,1] = PR[GP1:90,1] + 47.784;
   1:  PR[GP1:91,2] = PR[GP1:90,2] + -31.934;
   1:L PR[91] 10mm/sec CNT100;
   1:  PR[GP1:91,1] = PR[GP1:90,1] + 51.324;
   1:  PR[GP1:91,2] = PR[GP1:90,2] + -30.646;
   1:L PR[91] 10mm/sec CNT100;
   1:  PR[GP1:91,1] = PR[GP1:90,1] + 53.373;
   1:  PR[GP1:91,2] = PR[GP1:90,2] + -29.392;
   1:L PR[91] 10mm/sec CNT100;
   1:  PR[GP1:91,1] = PR[GP1:90,1] + 61.179;
   1:  PR[GP1:91,2] = PR[GP1:90,2] + -22.912;
   1:L PR[91] 10mm/sec CNT100;
   1:  PR[GP1:91,1] = PR[GP1:90,1] + 61.901;
   1:  PR[GP1:91,2] = PR[GP1:90,2] + -22.210;
   1:L PR[91] 10mm/sec CNT100;
   1:  PR[GP1:91,1] = PR[GP1:90,1] + 68.168;
   1:  PR[GP1:91,2] = PR[GP1:90,2] + -11.698;
   1:L PR[91] 10mm/sec CNT100;
   1:  PR[GP1:91,1] = PR[GP1:90,1] + 70.322;
   1:  PR[GP1:91,2] = PR[GP1:90,2] + 0.279;
   1:L PR[91] 10mm/sec CNT100;
   1:  PR[GP1:91,1] = PR[GP1:90,1] + 68.168;
   1:  PR[GP1:91,2] = PR[GP1:90,2] + 12.257;
   1:L PR[91] 10mm/sec CNT100;
   1:  PR[GP1:91,1] = PR[GP1:90,1] + 62.349;
   1:  PR[GP1:91,2] = PR[GP1:90,2] + 22.078;
   1:L PR[91] 10mm/sec CNT100;
   1:  PR[GP1:91,1] = PR[GP1:90,1] + 61.909;
   1:  PR[GP1:91,2] = PR[GP1:90,2] + 22.760;
   1:L PR[91] 10mm/sec CNT100;
   1:  PR[GP1:91,1] = PR[GP1:90,1] + 61.179;
   1:  PR[GP1:91,2] = PR[GP1:90,2] + 23.470;
   1:L PR[91] 10mm/sec CNT100;
   1:  PR[GP1:91,1] = PR[GP1:90,1] + 53.373;
   1:  PR[GP1:91,2] = PR[GP1:90,2] + 29.950;
   1:L PR[91] 10mm/sec CNT100;
   1:  PR[GP1:91,1] = PR[GP1:90,1] + 51.323;
   1:  PR[GP1:91,2] = PR[GP1:90,2] + 31.204;
   1:L PR[91] 10mm/sec CNT100;
   1:  PR[GP1:91,1] = PR[GP1:90,1] + 44.569;
   1:  PR[GP1:91,2] = PR[GP1:90,2] + 33.705;
   1:L PR[91] 10mm/sec CNT100;
   1:  PR[GP1:91,1] = PR[GP1:90,1] + 41.092;
   1:  PR[GP1:91,2] = PR[GP1:90,2] + 34.963;
   1:L PR[91] 10mm/sec CNT100;
   1:  PR[GP1:91,1] = PR[GP1:90,1] + 35.515;
   1:  PR[GP1:91,2] = PR[GP1:90,2] + 35.662;
   1:L PR[91] 10mm/sec CNT100;
   1:  PR[GP1:91,1] = PR[GP1:90,1] + 32.296;
   1:  PR[GP1:91,2] = PR[GP1:90,2] + 35.756;
   1:L PR[91] 10mm/sec CNT100;
   1:  PR[GP1:91,1] = PR[GP1:90,1] + 25.462;
   1:  PR[GP1:91,2] = PR[GP1:90,2] + 35.168;
   1:L PR[91] 10mm/sec CNT100;
   1:  PR[GP1:91,1] = PR[GP1:90,1] + 17.336;
   1:  PR[GP1:91,2] = PR[GP1:90,2] + 32.826;
   1:L PR[91] 10mm/sec CNT100;
   1:  PR[GP1:91,1] = PR[GP1:90,1] + 10.565;
   1:  PR[GP1:91,2] = PR[GP1:90,2] + 29.172;
   1:L PR[91] 10mm/sec CNT100;
   1:  PR[GP1:91,1] = PR[GP1:90,1] + 8.732;
   1:  PR[GP1:91,2] = PR[GP1:90,2] + 27.682;
   1:L PR[91] 10mm/sec CNT100;
   1:  PR[GP1:91,1] = PR[GP1:90,1] + 4.240;
   1:  PR[GP1:91,2] = PR[GP1:90,2] + 23.725;
   1:L PR[91] 10mm/sec CNT100;
   1:  PR[GP1:91,1] = PR[GP1:90,1] + 2.509;
   1:  PR[GP1:91,2] = PR[GP1:90,2] + 21.615;
   1:L PR[91] 10mm/sec CNT100;
   1:  PR[GP1:91,1] = PR[GP1:90,1] + 0.856;
   1:  PR[GP1:91,2] = PR[GP1:90,2] + 19.290;
   1:L PR[91] 10mm/sec CNT100;
   1:  PR[GP1:91,1] = PR[GP1:90,1] + -1.373;
   1:L PR[91] 10mm/sec CNT100;
   1:  PR[GP1:91,1] = PR[GP1:90,1] + -3.035;
   1:  PR[GP1:91,2] = PR[GP1:90,2] + 21.634;
   1:L PR[91] 10mm/sec CNT100;
   1:  PR[GP1:91,1] = PR[GP1:90,1] + -4.733;
   1:  PR[GP1:91,2] = PR[GP1:90,2] + 23.697;
   1:L PR[91] 10mm/sec CNT100;
   1:  PR[GP1:91,1] = PR[GP1:90,1] + -9.230;
   1:  PR[GP1:91,2] = PR[GP1:90,2] + 27.656;
   1:L PR[91] 10mm/sec CNT100;
   1:  PR[GP1:91,1] = PR[GP1:90,1] + -11.061;
   1:  PR[GP1:91,2] = PR[GP1:90,2] + 29.145;
   1:L PR[91] 10mm/sec CNT100;
   1:  PR[GP1:91,1] = PR[GP1:90,1] + -17.870;
   1:  PR[GP1:91,2] = PR[GP1:90,2] + 32.830;
   1:L PR[91] 10mm/sec CNT100;
   1:  PR[GP1:91,1] = PR[GP1:90,1] + -25.985;
   1:  PR[GP1:91,2] = PR[GP1:90,2] + 35.169;
   1:L PR[91] 10mm/sec CNT100;
   1:  PR[GP1:91,1] = PR[GP1:90,1] + -32.838;
   1:  PR[GP1:91,2] = PR[GP1:90,2] + 35.755;
   1:L PR[91] 10mm/sec CNT100;
   1:  PR[GP1:91,1] = PR[GP1:90,1] + -36.061;
   1:  PR[GP1:91,2] = PR[GP1:90,2] + 35.661;
   1:L PR[91] 10mm/sec CNT100;
   1:  PR[GP1:91,1] = PR[GP1:90,1] + -41.642;
   1:  PR[GP1:91,2] = PR[GP1:90,2] + 34.959;
   1:L PR[91] 10mm/sec CNT100;
   1:  PR[GP1:91,1] = PR[GP1:90,1] + -51.862;
   1:  PR[GP1:91,2] = PR[GP1:90,2] + 31.196;
   1:L PR[91] 10mm/sec CNT100;
   1:  PR[GP1:91,1] = PR[GP1:90,1] + -53.918;
   1:  PR[GP1:91,2] = PR[GP1:90,2] + 29.931;
   1:L PR[91] 10mm/sec CNT100;
   1:  PR[GP1:91,1] = PR[GP1:90,1] + -61.718;
   1:  PR[GP1:91,2] = PR[GP1:90,2] + 23.466;
   1:L PR[91] 10mm/sec CNT100;
   1:  PR[GP1:91,1] = PR[GP1:90,1] + -62.437;
   1:  PR[GP1:91,2] = PR[GP1:90,2] + 22.766;
   1:L PR[91] 10mm/sec CNT100;
   1:  PR[GP1:91,1] = PR[GP1:90,1] + -68.695;
   1:  PR[GP1:91,2] = PR[GP1:90,2] + 12.235;
   1:L PR[91] 10mm/sec CNT100;
   1:  PR[GP1:91,1] = PR[GP1:90,1] + -70.848;
   1:  PR[GP1:91,2] = PR[GP1:90,2] + 0.282;
   1:L PR[91] 10mm/sec CNT100;
   1:  PR[GP1:91,1] = PR[GP1:90,1] + -70.749;
   1:  PR[GP1:91,2] = PR[GP1:90,2] + -0.235;
   1:L PR[91] 10mm/sec CNT100;
   1:  PR[GP1:91,1] = PR[GP1:90,1] + -68.865;
   1:  PR[GP1:91,2] = PR[GP1:90,2] + -10.778;
   1:L PR[91] 10mm/sec CNT100;
   1:  PR[GP1:91,1] = PR[GP1:90,1] + -68.696;
   1:  PR[GP1:91,2] = PR[GP1:90,2] + -11.675;
   1:L PR[91] 10mm/sec CNT100;
   1:  PR[GP1:91,1] = PR[GP1:90,1] + -62.878;
   1:  PR[GP1:91,2] = PR[GP1:90,2] + -21.524;
   1:L PR[91] 10mm/sec CNT100;
   1:  PR[GP1:91,1] = PR[GP1:90,1] + -62.444;
   1:  PR[GP1:91,2] = PR[GP1:90,2] + -22.201;
   1:L PR[91] 10mm/sec CNT100;
   1:  PR[GP1:91,1] = PR[GP1:90,1] + -61.718;
   1:  PR[GP1:91,2] = PR[GP1:90,2] + -22.908;
   1:L PR[91] 10mm/sec CNT100;
   1:  PR[GP1:91,1] = PR[GP1:90,1] + -53.918;
   1:  PR[GP1:91,2] = PR[GP1:90,2] + -29.373;
   1:L PR[91] 10mm/sec CNT100;
   1:  PR[GP1:91,1] = PR[GP1:90,1] + -51.861;
   1:  PR[GP1:91,2] = PR[GP1:90,2] + -30.638;
   1:L PR[91] 10mm/sec CNT100;
   1:  PR[GP1:91,1] = PR[GP1:90,1] + -45.110;
   1:  PR[GP1:91,2] = PR[GP1:90,2] + -33.141;
   1:L PR[91] 10mm/sec CNT100;
   1:  PR[GP1:91,1] = PR[GP1:90,1] + -41.644;
   1:  PR[GP1:91,2] = PR[GP1:90,2] + -34.401;
   1:L PR[91] 10mm/sec CNT100;
   1:  PR[GP1:91,1] = PR[GP1:90,1] + -36.061;
   1:  PR[GP1:91,2] = PR[GP1:90,2] + -35.103;
   1:L PR[91] 10mm/sec CNT100;
   1:  PR[GP1:91,1] = PR[GP1:90,1] + -32.838;
   1:  PR[GP1:91,2] = PR[GP1:90,2] + -35.197;
   1:L PR[91] 10mm/sec CNT100;
   1:  PR[GP1:91,1] = PR[GP1:90,1] + -25.985;
   1:  PR[GP1:91,2] = PR[GP1:90,2] + -34.611;
   1:L PR[91] 10mm/sec CNT100;
   1:  PR[GP1:91,1] = PR[GP1:90,1] + -17.890;
   1:  PR[GP1:91,2] = PR[GP1:90,2] + -32.281;
   1:L PR[91] 10mm/sec CNT100;
   1:  PR[GP1:91,1] = PR[GP1:90,1] + -17.467;
   1:  PR[GP1:91,2] = PR[GP1:90,2] + -32.033;
   1:L PR[91] 10mm/sec CNT100;
   1:  PR[GP1:91,1] = PR[GP1:90,1] + -10.638;
   1:  PR[GP1:91,2] = PR[GP1:90,2] + -28.315;
   1:L PR[91] 10mm/sec CNT100;
   1:  PR[GP1:91,1] = PR[GP1:90,1] + -9.257;
   1:  PR[GP1:91,2] = PR[GP1:90,2] + -27.123;
   1:L PR[91] 10mm/sec CNT100;
   1:  PR[GP1:91,1] = PR[GP1:90,1] + -4.744;
   1:  PR[GP1:91,2] = PR[GP1:90,2] + -23.151;
   1:L PR[91] 10mm/sec CNT100;
   1:  PR[GP1:91,1] = PR[GP1:90,1] + -3.047;
   1:  PR[GP1:91,2] = PR[GP1:90,2] + -21.091;
   1:L PR[91] 10mm/sec CNT100;
   1:  PR[GP1:91,1] = PR[GP1:90,1] + -1.374;
   1:  PR[GP1:91,2] = PR[GP1:90,2] + -18.732;
   1:L PR[91] 10mm/sec CNT100;
   1:  PR[GP1:91,1] = PR[GP1:90,1] + 0.859;
   1:L PR[91] 10mm/sec CNT100;
   1:  PR[GP1:91,1] = PR[GP1:90,1] + 2.114;
   1:  PR[GP1:91,2] = PR[GP1:90,2] + -20.944;
   1:  PR[GP1:91,3] = PR[GP1:90,3] + 43.615;
   1:L PR[91] 10mm/sec CNT100;
   1:  PR[GP1:91,1] = PR[GP1:90,1] + 4.024;
   1:  PR[GP1:91,2] = PR[GP1:90,2] + -23.266;
   1:L PR[91] 10mm/sec CNT100;
   1:  PR[GP1:91,1] = PR[GP1:90,1] + 8.278;
   1:  PR[GP1:91,2] = PR[GP1:90,2] + -27.012;
   1:L PR[91] 10mm/sec CNT100;
   1:  PR[GP1:91,1] = PR[GP1:90,1] + 9.896;
   1:  PR[GP1:91,2] = PR[GP1:90,2] + -28.410;
   1:L PR[91] 10mm/sec CNT100;
   1:  PR[GP1:91,1] = PR[GP1:90,1] + 16.522;
   1:  PR[GP1:91,2] = PR[GP1:90,2] + -32.007;
   1:L PR[91] 10mm/sec CNT100;
   1:  PR[GP1:91,1] = PR[GP1:90,1] + 17.102;
   1:  PR[GP1:91,2] = PR[GP1:90,2] + -32.346;
   1:L PR[91] 10mm/sec CNT100;
   1:  PR[GP1:91,1] = PR[GP1:90,1] + 25.245;
   1:  PR[GP1:91,2] = PR[GP1:90,2] + -34.676;
   1:L PR[91] 10mm/sec CNT100;
   1:  PR[GP1:91,1] = PR[GP1:90,1] + 27.087;
   1:  PR[GP1:91,2] = PR[GP1:90,2] + -34.798;
   1:L PR[91] 10mm/sec CNT100;
   1:  PR[GP1:91,1] = PR[GP1:90,1] + 32.487;
   1:  PR[GP1:91,2] = PR[GP1:90,2] + -35.263;
   1:L PR[91] 10mm/sec CNT100;
   1:  PR[GP1:91,1] = PR[GP1:90,1] + 34.808;
   1:  PR[GP1:91,2] = PR[GP1:90,2] + -35.195;
   1:L PR[91] 10mm/sec CNT100;
   1:  PR[GP1:91,1] = PR[GP1:90,1] + 41.010;
   1:  PR[GP1:91,2] = PR[GP1:90,2] + -34.418;
   1:L PR[91] 10mm/sec CNT100;
   1:  PR[GP1:91,1] = PR[GP1:90,1] + 46.750;
   1:  PR[GP1:91,2] = PR[GP1:90,2] + -32.298;
   1:L PR[91] 10mm/sec CNT100;
   1:  PR[GP1:91,1] = PR[GP1:90,1] + 50.978;
   1:  PR[GP1:91,2] = PR[GP1:90,2] + -30.759;
   1:L PR[91] 10mm/sec CNT100;
   1:  PR[GP1:91,1] = PR[GP1:90,1] + 53.436;
   1:  PR[GP1:91,2] = PR[GP1:90,2] + -29.256;
   1:L PR[91] 10mm/sec CNT100;
   1:  PR[GP1:91,1] = PR[GP1:90,1] + 60.651;
   1:  PR[GP1:91,2] = PR[GP1:90,2] + -23.266;
   1:L PR[91] 10mm/sec CNT100;
   1:  PR[GP1:91,1] = PR[GP1:90,1] + 61.750;
   1:  PR[GP1:91,2] = PR[GP1:90,2] + -22.199;
   1:L PR[91] 10mm/sec CNT100;
   1:  PR[GP1:91,1] = PR[GP1:90,1] + 67.648;
   1:  PR[GP1:91,2] = PR[GP1:90,2] + -12.303;
   1:L PR[91] 10mm/sec CNT100;
   1:  PR[GP1:91,1] = PR[GP1:90,1] + 67.942;
   1:  PR[GP1:91,2] = PR[GP1:90,2] + -11.841;
   1:L PR[91] 10mm/sec CNT100;
   1:  PR[GP1:91,1] = PR[GP1:90,1] + 68.069;
   1:  PR[GP1:91,2] = PR[GP1:90,2] + -11.499;
   1:L PR[91] 10mm/sec CNT100;
   1:  PR[GP1:91,1] = PR[GP1:90,1] + 70.202;
   1:  PR[GP1:91,2] = PR[GP1:90,2] + 0.278;
   1:L PR[91] 10mm/sec CNT100;
   1:  PR[GP1:91,1] = PR[GP1:90,1] + 68.106;
   1:  PR[GP1:91,2] = PR[GP1:90,2] + 11.677;
   1:L PR[91] 10mm/sec CNT100;
   1:  PR[GP1:91,1] = PR[GP1:90,1] + 68.061;
   1:  PR[GP1:91,2] = PR[GP1:90,2] + 12.076;
   1:L PR[91] 10mm/sec CNT100;
   1:  PR[GP1:91,1] = PR[GP1:90,1] + 67.938;
   1:  PR[GP1:91,2] = PR[GP1:90,2] + 12.409;
   1:L PR[91] 10mm/sec CNT100;
   1:  PR[GP1:91,1] = PR[GP1:90,1] + 62.425;
   1:  PR[GP1:91,2] = PR[GP1:90,2] + 21.713;
   1:L PR[91] 10mm/sec CNT100;
   1:  PR[GP1:91,1] = PR[GP1:90,1] + 61.757;
   1:  PR[GP1:91,2] = PR[GP1:90,2] + 22.749;
   1:L PR[91] 10mm/sec CNT100;
   1:  PR[GP1:91,1] = PR[GP1:90,1] + 60.651;
   1:  PR[GP1:91,2] = PR[GP1:90,2] + 23.824;
   1:L PR[91] 10mm/sec CNT100;
   1:  PR[GP1:91,1] = PR[GP1:90,1] + 53.436;
   1:  PR[GP1:91,2] = PR[GP1:90,2] + 29.814;
   1:L PR[91] 10mm/sec CNT100;
   1:  PR[GP1:91,1] = PR[GP1:90,1] + 50.977;
   1:  PR[GP1:91,2] = PR[GP1:90,2] + 31.318;
   1:L PR[91] 10mm/sec CNT100;
   1:  PR[GP1:91,1] = PR[GP1:90,1] + 44.880;
   1:  PR[GP1:91,2] = PR[GP1:90,2] + 33.576;
   1:L PR[91] 10mm/sec CNT100;
   1:  PR[GP1:91,1] = PR[GP1:90,1] + 41.012;
   1:  PR[GP1:91,2] = PR[GP1:90,2] + 34.976;
   1:L PR[91] 10mm/sec CNT100;
   1:  PR[GP1:91,1] = PR[GP1:90,1] + 34.808;
   1:  PR[GP1:91,2] = PR[GP1:90,2] + 35.753;
   1:L PR[91] 10mm/sec CNT100;
   1:  PR[GP1:91,1] = PR[GP1:90,1] + 32.487;
   1:  PR[GP1:91,2] = PR[GP1:90,2] + 35.821;
   1:L PR[91] 10mm/sec CNT100;
   1:  PR[GP1:91,1] = PR[GP1:90,1] + 27.087;
   1:  PR[GP1:91,2] = PR[GP1:90,2] + 35.356;
   1:L PR[91] 10mm/sec CNT100;
   1:  PR[GP1:91,1] = PR[GP1:90,1] + 25.243;
   1:  PR[GP1:91,2] = PR[GP1:90,2] + 35.234;
   1:L PR[91] 10mm/sec CNT100;
   1:  PR[GP1:91,1] = PR[GP1:90,1] + 17.077;
   1:  PR[GP1:91,2] = PR[GP1:90,2] + 32.894;
   1:L PR[91] 10mm/sec CNT100;
   1:  PR[GP1:91,1] = PR[GP1:90,1] + 10.392;
   1:  PR[GP1:91,2] = PR[GP1:90,2] + 29.286;
   1:L PR[91] 10mm/sec CNT100;
   1:  PR[GP1:91,1] = PR[GP1:90,1] + 8.248;
   1:  PR[GP1:91,2] = PR[GP1:90,2] + 27.542;
   1:L PR[91] 10mm/sec CNT100;
   1:  PR[GP1:91,1] = PR[GP1:90,1] + 4.011;
   1:  PR[GP1:91,2] = PR[GP1:90,2] + 23.811;
   1:L PR[91] 10mm/sec CNT100;
   1:  PR[GP1:91,1] = PR[GP1:90,1] + 2.072;
   1:  PR[GP1:91,2] = PR[GP1:90,2] + 21.446;
   1:L PR[91] 10mm/sec CNT100;
   1:  PR[GP1:91,1] = PR[GP1:90,1] + 0.769;
   1:  PR[GP1:91,2] = PR[GP1:90,2] + 19.615;
   1:L PR[91] 10mm/sec CNT100;
   1:  PR[GP1:91,1] = PR[GP1:90,1] + -1.286;
   1:L PR[91] 10mm/sec CNT100;
   1:  PR[GP1:91,1] = PR[GP1:90,1] + -2.604;
   1:  PR[GP1:91,2] = PR[GP1:90,2] + 21.473;
   1:L PR[91] 10mm/sec CNT100;
   1:  PR[GP1:91,1] = PR[GP1:90,1] + -4.506;
   1:  PR[GP1:91,2] = PR[GP1:90,2] + 23.784;
   1:L PR[91] 10mm/sec CNT100;
   1:  PR[GP1:91,1] = PR[GP1:90,1] + -8.747;
   1:  PR[GP1:91,2] = PR[GP1:90,2] + 27.518;
   1:L PR[91] 10mm/sec CNT100;
   1:  PR[GP1:91,1] = PR[GP1:90,1] + -10.889;
   1:  PR[GP1:91,2] = PR[GP1:90,2] + 29.259;
   1:L PR[91] 10mm/sec CNT100;
   1:  PR[GP1:91,1] = PR[GP1:90,1] + -17.611;
   1:  PR[GP1:91,2] = PR[GP1:90,2] + 32.898;
   1:L PR[91] 10mm/sec CNT100;
   1:  PR[GP1:91,1] = PR[GP1:90,1] + -25.767;
   1:  PR[GP1:91,2] = PR[GP1:90,2] + 35.234;
   1:L PR[91] 10mm/sec CNT100;
   1:  PR[GP1:91,1] = PR[GP1:90,1] + -27.613;
   1:  PR[GP1:91,2] = PR[GP1:90,2] + 35.356;
   1:L PR[91] 10mm/sec CNT100;
   1:  PR[GP1:91,1] = PR[GP1:90,1] + -33.029;
   1:  PR[GP1:91,2] = PR[GP1:90,2] + 35.820;
   1:L PR[91] 10mm/sec CNT100;
   1:  PR[GP1:91,1] = PR[GP1:90,1] + -35.355;
   1:  PR[GP1:91,2] = PR[GP1:90,2] + 35.752;
   1:L PR[91] 10mm/sec CNT100;
   1:  PR[GP1:91,1] = PR[GP1:90,1] + -41.564;
   1:  PR[GP1:91,2] = PR[GP1:90,2] + 34.971;
   1:L PR[91] 10mm/sec CNT100;
   1:  PR[GP1:91,1] = PR[GP1:90,1] + -47.307;
   1:  PR[GP1:91,2] = PR[GP1:90,2] + 32.847;
   1:L PR[91] 10mm/sec CNT100;
   1:  PR[GP1:91,1] = PR[GP1:90,1] + -51.518;
   1:  PR[GP1:91,2] = PR[GP1:90,2] + 31.308;
   1:L PR[91] 10mm/sec CNT100;
   1:  PR[GP1:91,1] = PR[GP1:90,1] + -53.984;
   1:  PR[GP1:91,2] = PR[GP1:90,2] + 29.792;
   1:L PR[91] 10mm/sec CNT100;
   1:  PR[GP1:91,1] = PR[GP1:90,1] + -61.194;
   1:  PR[GP1:91,2] = PR[GP1:90,2] + 23.816;
   1:L PR[91] 10mm/sec CNT100;
   1:  PR[GP1:91,1] = PR[GP1:90,1] + -62.289;
   1:  PR[GP1:91,2] = PR[GP1:90,2] + 22.750;
   1:L PR[91] 10mm/sec CNT100;
   1:  PR[GP1:91,1] = PR[GP1:90,1] + -68.180;
   1:  PR[GP1:91,2] = PR[GP1:90,2] + 12.835;
   1:L PR[91] 10mm/sec CNT100;
   1:  PR[GP1:91,1] = PR[GP1:90,1] + -68.469;
   1:  PR[GP1:91,2] = PR[GP1:90,2] + 12.378;
   1:L PR[91] 10mm/sec CNT100;
   1:  PR[GP1:91,1] = PR[GP1:90,1] + -68.597;
   1:  PR[GP1:91,2] = PR[GP1:90,2] + 12.028;
   1:L PR[91] 10mm/sec CNT100;
   1:  PR[GP1:91,1] = PR[GP1:90,1] + -70.728;
   1:  PR[GP1:91,2] = PR[GP1:90,2] + 0.280;
   1:L PR[91] 10mm/sec CNT100;
   1:  PR[GP1:91,1] = PR[GP1:90,1] + -68.632;
   1:  PR[GP1:91,2] = PR[GP1:90,2] + -11.099;
   1:L PR[91] 10mm/sec CNT100;
   1:  PR[GP1:91,1] = PR[GP1:90,1] + -68.590;
   1:  PR[GP1:91,2] = PR[GP1:90,2] + -11.490;
   1:L PR[91] 10mm/sec CNT100;
   1:  PR[GP1:91,1] = PR[GP1:90,1] + -68.466;
   1:  PR[GP1:91,2] = PR[GP1:90,2] + -11.829;
   1:L PR[91] 10mm/sec CNT100;
   1:  PR[GP1:91,1] = PR[GP1:90,1] + -62.955;
   1:  PR[GP1:91,2] = PR[GP1:90,2] + -21.156;
   1:L PR[91] 10mm/sec CNT100;
   1:  PR[GP1:91,1] = PR[GP1:90,1] + -62.296;
   1:  PR[GP1:91,2] = PR[GP1:90,2] + -22.185;
   1:L PR[91] 10mm/sec CNT100;
   1:  PR[GP1:91,1] = PR[GP1:90,1] + -61.194;
   1:  PR[GP1:91,2] = PR[GP1:90,2] + -23.258;
   1:L PR[91] 10mm/sec CNT100;
   1:  PR[GP1:91,1] = PR[GP1:90,1] + -53.984;
   1:  PR[GP1:91,2] = PR[GP1:90,2] + -29.234;
   1:L PR[91] 10mm/sec CNT100;
   1:  PR[GP1:91,1] = PR[GP1:90,1] + -51.517;
   1:  PR[GP1:91,2] = PR[GP1:90,2] + -30.751;
   1:L PR[91] 10mm/sec CNT100;
   1:  PR[GP1:91,1] = PR[GP1:90,1] + -45.422;
   1:  PR[GP1:91,2] = PR[GP1:90,2] + -33.011;
   1:L PR[91] 10mm/sec CNT100;
   1:  PR[GP1:91,1] = PR[GP1:90,1] + -41.565;
   1:  PR[GP1:91,2] = PR[GP1:90,2] + -34.412;
   1:L PR[91] 10mm/sec CNT100;
   1:  PR[GP1:91,1] = PR[GP1:90,1] + -35.355;
   1:  PR[GP1:91,2] = PR[GP1:90,2] + -35.194;
   1:L PR[91] 10mm/sec CNT100;
   1:  PR[GP1:91,1] = PR[GP1:90,1] + -33.029;
   1:  PR[GP1:91,2] = PR[GP1:90,2] + -35.262;
   1:L PR[91] 10mm/sec CNT100;
   1:  PR[GP1:91,1] = PR[GP1:90,1] + -27.613;
   1:  PR[GP1:91,2] = PR[GP1:90,2] + -34.798;
   1:L PR[91] 10mm/sec CNT100;
   1:  PR[GP1:91,1] = PR[GP1:90,1] + -25.768;
   1:  PR[GP1:91,2] = PR[GP1:90,2] + -34.676;
   1:L PR[91] 10mm/sec CNT100;
   1:  PR[GP1:91,1] = PR[GP1:90,1] + -17.635;
   1:  PR[GP1:91,2] = PR[GP1:90,2] + -32.350;
   1:L PR[91] 10mm/sec CNT100;
   1:  PR[GP1:91,1] = PR[GP1:90,1] + -17.056;
   1:  PR[GP1:91,2] = PR[GP1:90,2] + -32.011;
   1:L PR[91] 10mm/sec CNT100;
   1:  PR[GP1:91,1] = PR[GP1:90,1] + -10.394;
   1:  PR[GP1:91,2] = PR[GP1:90,2] + -28.384;
   1:L PR[91] 10mm/sec CNT100;
   1:  PR[GP1:91,1] = PR[GP1:90,1] + -8.777;
   1:  PR[GP1:91,2] = PR[GP1:90,2] + -26.988;
   1:L PR[91] 10mm/sec CNT100;
   1:  PR[GP1:91,1] = PR[GP1:90,1] + -4.518;
   1:  PR[GP1:91,2] = PR[GP1:90,2] + -23.239;
   1:L PR[91] 10mm/sec CNT100;
   1:  PR[GP1:91,1] = PR[GP1:90,1] + -2.616;
   1:  PR[GP1:91,2] = PR[GP1:90,2] + -20.932;
   1:L PR[91] 10mm/sec CNT100;
   1:  PR[GP1:91,1] = PR[GP1:90,1] + -1.287;
   1:  PR[GP1:91,2] = PR[GP1:90,2] + -19.057;
   1:L PR[91] 10mm/sec CNT100;
   1:  PR[GP1:91,1] = PR[GP1:90,1] + 0.773;
   1:L PR[91] 10mm/sec CNT100;
   1:  PR[GP1:91,1] = PR[GP1:90,1] + 1.681;
   1:  PR[GP1:91,2] = PR[GP1:90,2] + -20.781;
   1:  PR[GP1:91,3] = PR[GP1:90,3] + 44.225;
   1:L PR[91] 10mm/sec CNT100;
   1:  PR[GP1:91,1] = PR[GP1:90,1] + 3.797;
   1:  PR[GP1:91,2] = PR[GP1:90,2] + -23.353;
   1:L PR[91] 10mm/sec CNT100;
   1:  PR[GP1:91,1] = PR[GP1:90,1] + 7.796;
   1:  PR[GP1:91,2] = PR[GP1:90,2] + -26.875;
   1:L PR[91] 10mm/sec CNT100;
   1:  PR[GP1:91,1] = PR[GP1:90,1] + 9.652;
   1:  PR[GP1:91,2] = PR[GP1:90,2] + -28.479;
   1:L PR[91] 10mm/sec CNT100;
   1:  PR[GP1:91,1] = PR[GP1:90,1] + 16.111;
   1:  PR[GP1:91,2] = PR[GP1:90,2] + -31.985;
   1:L PR[91] 10mm/sec CNT100;
   1:  PR[GP1:91,1] = PR[GP1:90,1] + 16.847;
   1:  PR[GP1:91,2] = PR[GP1:90,2] + -32.416;
   1:L PR[91] 10mm/sec CNT100;
   1:  PR[GP1:91,1] = PR[GP1:90,1] + 24.759;
   1:  PR[GP1:91,2] = PR[GP1:90,2] + -34.688;
   1:L PR[91] 10mm/sec CNT100;
   1:  PR[GP1:91,1] = PR[GP1:90,1] + 25.052;
   1:  PR[GP1:91,2] = PR[GP1:90,2] + -34.755;
   1:L PR[91] 10mm/sec CNT100;
   1:  PR[GP1:91,1] = PR[GP1:90,1] + 29.325;
   1:  PR[GP1:91,2] = PR[GP1:90,2] + -35.039;
   1:L PR[91] 10mm/sec CNT100;
   1:  PR[GP1:91,1] = PR[GP1:90,1] + 32.678;
   1:  PR[GP1:91,2] = PR[GP1:90,2] + -35.327;
   1:L PR[91] 10mm/sec CNT100;
   1:  PR[GP1:91,1] = PR[GP1:90,1] + 34.100;
   1:  PR[GP1:91,2] = PR[GP1:90,2] + -35.286;
   1:L PR[91] 10mm/sec CNT100;
   1:  PR[GP1:91,1] = PR[GP1:90,1] + 40.929;
   1:  PR[GP1:91,2] = PR[GP1:90,2] + -34.430;
   1:L PR[91] 10mm/sec CNT100;
   1:  PR[GP1:91,1] = PR[GP1:90,1] + 45.716;
   1:  PR[GP1:91,2] = PR[GP1:90,2] + -32.663;
   1:L PR[91] 10mm/sec CNT100;
   1:  PR[GP1:91,1] = PR[GP1:90,1] + 50.632;
   1:  PR[GP1:91,2] = PR[GP1:90,2] + -30.873;
   1:L PR[91] 10mm/sec CNT100;
   1:  PR[GP1:91,1] = PR[GP1:90,1] + 53.498;
   1:  PR[GP1:91,2] = PR[GP1:90,2] + -29.120;
   1:L PR[91] 10mm/sec CNT100;
   1:  PR[GP1:91,1] = PR[GP1:90,1] + 60.123;
   1:  PR[GP1:91,2] = PR[GP1:90,2] + -23.620;
   1:L PR[91] 10mm/sec CNT100;
   1:  PR[GP1:91,1] = PR[GP1:90,1] + 61.598;
   1:  PR[GP1:91,2] = PR[GP1:90,2] + -22.187;
   1:L PR[91] 10mm/sec CNT100;
   1:  PR[GP1:91,1] = PR[GP1:90,1] + 67.093;
   1:  PR[GP1:91,2] = PR[GP1:90,2] + -12.967;
   1:L PR[91] 10mm/sec CNT100;
   1:  PR[GP1:91,1] = PR[GP1:90,1] + 67.684;
   1:  PR[GP1:91,2] = PR[GP1:90,2] + -12.039;
   1:L PR[91] 10mm/sec CNT100;
   1:  PR[GP1:91,1] = PR[GP1:90,1] + 67.965;
   1:  PR[GP1:91,2] = PR[GP1:90,2] + -11.281;
   1:L PR[91] 10mm/sec CNT100;
   1:  PR[GP1:91,1] = PR[GP1:90,1] + 69.992;
   1:  PR[GP1:91,2] = PR[GP1:90,2] + -0.091;
   1:L PR[91] 10mm/sec CNT100;
   1:  PR[GP1:91,1] = PR[GP1:90,1] + 70.032;
   1:  PR[GP1:91,2] = PR[GP1:90,2] + 0.258;
   1:L PR[91] 10mm/sec CNT100;
   1:  PR[GP1:91,1] = PR[GP1:90,1] + 68.048;
   1:  PR[GP1:91,2] = PR[GP1:90,2] + 11.044;
   1:L PR[91] 10mm/sec CNT100;
   1:  PR[GP1:91,1] = PR[GP1:90,1] + 67.958;
   1:  PR[GP1:91,2] = PR[GP1:90,2] + 11.859;
   1:L PR[91] 10mm/sec CNT100;
   1:  PR[GP1:91,1] = PR[GP1:90,1] + 67.681;
   1:  PR[GP1:91,2] = PR[GP1:90,2] + 12.607;
   1:L PR[91] 10mm/sec CNT100;
   1:  PR[GP1:91,1] = PR[GP1:90,1] + 62.502;
   1:  PR[GP1:91,2] = PR[GP1:90,2] + 21.347;
   1:L PR[91] 10mm/sec CNT100;
   1:  PR[GP1:91,1] = PR[GP1:90,1] + 61.605;
   1:  PR[GP1:91,2] = PR[GP1:90,2] + 22.738;
   1:L PR[91] 10mm/sec CNT100;
   1:  PR[GP1:91,1] = PR[GP1:90,1] + 60.123;
   1:  PR[GP1:91,2] = PR[GP1:90,2] + 24.178;
   1:L PR[91] 10mm/sec CNT100;
   1:  PR[GP1:91,1] = PR[GP1:90,1] + 53.499;
   1:  PR[GP1:91,2] = PR[GP1:90,2] + 29.678;
   1:L PR[91] 10mm/sec CNT100;
   1:  PR[GP1:91,1] = PR[GP1:90,1] + 50.631;
   1:  PR[GP1:91,2] = PR[GP1:90,2] + 31.432;
   1:L PR[91] 10mm/sec CNT100;
   1:  PR[GP1:91,1] = PR[GP1:90,1] + 45.191;
   1:  PR[GP1:91,2] = PR[GP1:90,2] + 33.447;
   1:L PR[91] 10mm/sec CNT100;
   1:  PR[GP1:91,1] = PR[GP1:90,1] + 40.931;
   1:  PR[GP1:91,2] = PR[GP1:90,2] + 34.988;
   1:L PR[91] 10mm/sec CNT100;
   1:  PR[GP1:91,1] = PR[GP1:90,1] + 34.100;
   1:  PR[GP1:91,2] = PR[GP1:90,2] + 35.844;
   1:L PR[91] 10mm/sec CNT100;
   1:  PR[GP1:91,1] = PR[GP1:90,1] + 32.678;
   1:  PR[GP1:91,2] = PR[GP1:90,2] + 35.885;
   1:L PR[91] 10mm/sec CNT100;
   1:  PR[GP1:91,1] = PR[GP1:90,1] + 29.325;
   1:  PR[GP1:91,2] = PR[GP1:90,2] + 35.597;
   1:L PR[91] 10mm/sec CNT100;
   1:  PR[GP1:91,1] = PR[GP1:90,1] + 25.050;
   1:  PR[GP1:91,2] = PR[GP1:90,2] + 35.313;
   1:L PR[91] 10mm/sec CNT100;
   1:  PR[GP1:91,1] = PR[GP1:90,1] + 24.752;
   1:  PR[GP1:91,2] = PR[GP1:90,2] + 35.242;
   1:L PR[91] 10mm/sec CNT100;
   1:  PR[GP1:91,1] = PR[GP1:90,1] + 16.820;
   1:  PR[GP1:91,2] = PR[GP1:90,2] + 32.962;
   1:L PR[91] 10mm/sec CNT100;
   1:  PR[GP1:91,1] = PR[GP1:90,1] + 10.219;
   1:  PR[GP1:91,2] = PR[GP1:90,2] + 29.400;
   1:L PR[91] 10mm/sec CNT100;
   1:  PR[GP1:91,1] = PR[GP1:90,1] + 7.763;
   1:  PR[GP1:91,2] = PR[GP1:90,2] + 27.403;
   1:L PR[91] 10mm/sec CNT100;
   1:  PR[GP1:91,1] = PR[GP1:90,1] + 3.781;
   1:  PR[GP1:91,2] = PR[GP1:90,2] + 23.896;
   1:L PR[91] 10mm/sec CNT100;
   1:  PR[GP1:91,1] = PR[GP1:90,1] + 1.634;
   1:  PR[GP1:91,2] = PR[GP1:90,2] + 21.277;
   1:L PR[91] 10mm/sec CNT100;
   1:  PR[GP1:91,1] = PR[GP1:90,1] + 0.683;
   1:  PR[GP1:91,2] = PR[GP1:90,2] + 19.940;
   1:L PR[91] 10mm/sec CNT100;
   1:  PR[GP1:91,1] = PR[GP1:90,1] + -1.199;
   1:L PR[91] 10mm/sec CNT100;
   1:  PR[GP1:91,1] = PR[GP1:90,1] + -2.172;
   1:  PR[GP1:91,2] = PR[GP1:90,2] + 21.312;
   1:L PR[91] 10mm/sec CNT100;
   1:  PR[GP1:91,1] = PR[GP1:90,1] + -4.279;
   1:  PR[GP1:91,2] = PR[GP1:90,2] + 23.871;
   1:L PR[91] 10mm/sec CNT100;
   1:  PR[GP1:91,1] = PR[GP1:90,1] + -8.264;
   1:  PR[GP1:91,2] = PR[GP1:90,2] + 27.380;
   1:L PR[91] 10mm/sec CNT100;
   1:  PR[GP1:91,1] = PR[GP1:90,1] + -10.716;
   1:  PR[GP1:91,2] = PR[GP1:90,2] + 29.374;
   1:L PR[91] 10mm/sec CNT100;
   1:  PR[GP1:91,1] = PR[GP1:90,1] + -17.353;
   1:  PR[GP1:91,2] = PR[GP1:90,2] + 32.965;
   1:L PR[91] 10mm/sec CNT100;
   1:  PR[GP1:91,1] = PR[GP1:90,1] + -25.275;
   1:  PR[GP1:91,2] = PR[GP1:90,2] + 35.243;
   1:L PR[91] 10mm/sec CNT100;
   1:  PR[GP1:91,1] = PR[GP1:90,1] + -25.573;
   1:  PR[GP1:91,2] = PR[GP1:90,2] + 35.313;
   1:L PR[91] 10mm/sec CNT100;
   1:  PR[GP1:91,1] = PR[GP1:90,1] + -29.851;
   1:  PR[GP1:91,2] = PR[GP1:90,2] + 35.596;
   1:L PR[91] 10mm/sec CNT100;
   1:  PR[GP1:91,1] = PR[GP1:90,1] + -33.221;
   1:  PR[GP1:91,2] = PR[GP1:90,2] + 35.884;
   1:L PR[91] 10mm/sec CNT100;
   1:  PR[GP1:91,1] = PR[GP1:90,1] + -34.650;
   1:  PR[GP1:91,2] = PR[GP1:90,2] + 35.842;
   1:L PR[91] 10mm/sec CNT100;
   1:  PR[GP1:91,1] = PR[GP1:90,1] + -41.485;
   1:  PR[GP1:91,2] = PR[GP1:90,2] + 34.982;
   1:L PR[91] 10mm/sec CNT100;
   1:  PR[GP1:91,1] = PR[GP1:90,1] + -46.278;
   1:  PR[GP1:91,2] = PR[GP1:90,2] + 33.210;
   1:L PR[91] 10mm/sec CNT100;
   1:  PR[GP1:91,1] = PR[GP1:90,1] + -51.174;
   1:  PR[GP1:91,2] = PR[GP1:90,2] + 31.422;
   1:L PR[91] 10mm/sec CNT100;
   1:  PR[GP1:91,1] = PR[GP1:90,1] + -54.050;
   1:  PR[GP1:91,2] = PR[GP1:90,2] + 29.653;
   1:L PR[91] 10mm/sec CNT100;
   1:  PR[GP1:91,1] = PR[GP1:90,1] + -60.671;
   1:  PR[GP1:91,2] = PR[GP1:90,2] + 24.165;
   1:L PR[91] 10mm/sec CNT100;
   1:  PR[GP1:91,1] = PR[GP1:90,1] + -62.141;
   1:  PR[GP1:91,2] = PR[GP1:90,2] + 22.735;
   1:L PR[91] 10mm/sec CNT100;
   1:  PR[GP1:91,1] = PR[GP1:90,1] + -67.630;
   1:  PR[GP1:91,2] = PR[GP1:90,2] + 13.495;
   1:L PR[91] 10mm/sec CNT100;
   1:  PR[GP1:91,1] = PR[GP1:90,1] + -68.213;
   1:  PR[GP1:91,2] = PR[GP1:90,2] + 12.575;
   1:L PR[91] 10mm/sec CNT100;
   1:  PR[GP1:91,1] = PR[GP1:90,1] + -68.495;
   1:  PR[GP1:91,2] = PR[GP1:90,2] + 11.802;
   1:L PR[91] 10mm/sec CNT100;
   1:  PR[GP1:91,1] = PR[GP1:90,1] + -70.520;
   1:  PR[GP1:91,2] = PR[GP1:90,2] + 0.640;
   1:L PR[91] 10mm/sec CNT100;
   1:  PR[GP1:91,1] = PR[GP1:90,1] + -70.558;
   1:  PR[GP1:91,2] = PR[GP1:90,2] + 0.301;
   1:L PR[91] 10mm/sec CNT100;
   1:  PR[GP1:91,1] = PR[GP1:90,1] + -68.575;
   1:  PR[GP1:91,2] = PR[GP1:90,2] + -10.467;
   1:L PR[91] 10mm/sec CNT100;
   1:  PR[GP1:91,1] = PR[GP1:90,1] + -68.488;
   1:  PR[GP1:91,2] = PR[GP1:90,2] + -11.265;
   1:L PR[91] 10mm/sec CNT100;
   1:  PR[GP1:91,1] = PR[GP1:90,1] + -68.210;
   1:  PR[GP1:91,2] = PR[GP1:90,2] + -12.026;
   1:L PR[91] 10mm/sec CNT100;
   1:  PR[GP1:91,1] = PR[GP1:90,1] + -63.032;
   1:  PR[GP1:91,2] = PR[GP1:90,2] + -20.789;
   1:L PR[91] 10mm/sec CNT100;
   1:  PR[GP1:91,1] = PR[GP1:90,1] + -62.149;
   1:  PR[GP1:91,2] = PR[GP1:90,2] + -22.169;
   1:L PR[91] 10mm/sec CNT100;
   1:  PR[GP1:91,1] = PR[GP1:90,1] + -60.671;
   1:  PR[GP1:91,2] = PR[GP1:90,2] + -23.607;
   1:L PR[91] 10mm/sec CNT100;
   1:  PR[GP1:91,1] = PR[GP1:90,1] + -54.050;
   1:  PR[GP1:91,2] = PR[GP1:90,2] + -29.095;
   1:L PR[91] 10mm/sec CNT100;
   1:  PR[GP1:91,1] = PR[GP1:90,1] + -51.173;
   1:  PR[GP1:91,2] = PR[GP1:90,2] + -30.864;
   1:L PR[91] 10mm/sec CNT100;
   1:  PR[GP1:91,1] = PR[GP1:90,1] + -45.733;
   1:  PR[GP1:91,2] = PR[GP1:90,2] + -32.881;
   1:L PR[91] 10mm/sec CNT100;
   1:  PR[GP1:91,1] = PR[GP1:90,1] + -41.487;
   1:  PR[GP1:91,2] = PR[GP1:90,2] + -34.424;
   1:L PR[91] 10mm/sec CNT100;
   1:  PR[GP1:91,1] = PR[GP1:90,1] + -34.650;
   1:  PR[GP1:91,2] = PR[GP1:90,2] + -35.284;
   1:L PR[91] 10mm/sec CNT100;
   1:  PR[GP1:91,1] = PR[GP1:90,1] + -33.221;
   1:  PR[GP1:91,2] = PR[GP1:90,2] + -35.326;
   1:L PR[91] 10mm/sec CNT100;
   1:  PR[GP1:91,1] = PR[GP1:90,1] + -29.851;
   1:  PR[GP1:91,2] = PR[GP1:90,2] + -35.038;
   1:L PR[91] 10mm/sec CNT100;
   1:  PR[GP1:91,1] = PR[GP1:90,1] + -25.575;
   1:  PR[GP1:91,2] = PR[GP1:90,2] + -34.756;
   1:L PR[91] 10mm/sec CNT100;
   1:  PR[GP1:91,1] = PR[GP1:90,1] + -25.283;
   1:  PR[GP1:91,2] = PR[GP1:90,2] + -34.689;
   1:L PR[91] 10mm/sec CNT100;
   1:  PR[GP1:91,1] = PR[GP1:90,1] + -17.381;
   1:  PR[GP1:91,2] = PR[GP1:90,2] + -32.419;
   1:L PR[91] 10mm/sec CNT100;
   1:  PR[GP1:91,1] = PR[GP1:90,1] + -16.646;
   1:  PR[GP1:91,2] = PR[GP1:90,2] + -31.989;
   1:L PR[91] 10mm/sec CNT100;
   1:  PR[GP1:91,1] = PR[GP1:90,1] + -10.151;
   1:  PR[GP1:91,2] = PR[GP1:90,2] + -28.453;
   1:L PR[91] 10mm/sec CNT100;
   1:  PR[GP1:91,1] = PR[GP1:90,1] + -8.297;
   1:  PR[GP1:91,2] = PR[GP1:90,2] + -26.853;
   1:L PR[91] 10mm/sec CNT100;
   1:  PR[GP1:91,1] = PR[GP1:90,1] + -4.292;
   1:  PR[GP1:91,2] = PR[GP1:90,2] + -23.328;
   1:L PR[91] 10mm/sec CNT100;
   1:  PR[GP1:91,1] = PR[GP1:90,1] + -2.186;
   1:  PR[GP1:91,2] = PR[GP1:90,2] + -20.773;
   1:L PR[91] 10mm/sec CNT100;
   1:  PR[GP1:91,1] = PR[GP1:90,1] + -1.200;
   1:  PR[GP1:91,2] = PR[GP1:90,2] + -19.382;
   1:L PR[91] 10mm/sec CNT100;
   1:  PR[GP1:91,1] = PR[GP1:90,1] + 0.686;
   1:L PR[91] 10mm/sec CNT100;
   1:  PR[GP1:91,1] = PR[GP1:90,1] + 1.248;
   1:  PR[GP1:91,2] = PR[GP1:90,2] + -20.618;
   1:  PR[GP1:91,3] = PR[GP1:90,3] + 44.835;
   1:L PR[91] 10mm/sec CNT100;
   1:  PR[GP1:91,1] = PR[GP1:90,1] + 3.569;
   1:  PR[GP1:91,2] = PR[GP1:90,2] + -23.440;
   1:L PR[91] 10mm/sec CNT100;
   1:  PR[GP1:91,1] = PR[GP1:90,1] + 7.315;
   1:  PR[GP1:91,2] = PR[GP1:90,2] + -26.739;
   1:L PR[91] 10mm/sec CNT100;
   1:  PR[GP1:91,1] = PR[GP1:90,1] + 9.407;
   1:  PR[GP1:91,2] = PR[GP1:90,2] + -28.547;
   1:L PR[91] 10mm/sec CNT100;
   1:  PR[GP1:91,1] = PR[GP1:90,1] + 15.701;
   1:  PR[GP1:91,2] = PR[GP1:90,2] + -31.963;
   1:L PR[91] 10mm/sec CNT100;
   1:  PR[GP1:91,1] = PR[GP1:90,1] + 16.593;
   1:  PR[GP1:91,2] = PR[GP1:90,2] + -32.485;
   1:L PR[91] 10mm/sec CNT100;
   1:  PR[GP1:91,1] = PR[GP1:90,1] + 24.384;
   1:  PR[GP1:91,2] = PR[GP1:90,2] + -34.723;
   1:L PR[91] 10mm/sec CNT100;
   1:  PR[GP1:91,1] = PR[GP1:90,1] + 24.875;
   1:  PR[GP1:91,2] = PR[GP1:90,2] + -34.835;
   1:L PR[91] 10mm/sec CNT100;
   1:  PR[GP1:91,1] = PR[GP1:90,1] + 31.562;
   1:  PR[GP1:91,2] = PR[GP1:90,2] + -35.279;
   1:L PR[91] 10mm/sec CNT100;
   1:  PR[GP1:91,1] = PR[GP1:90,1] + 32.869;
   1:  PR[GP1:91,2] = PR[GP1:90,2] + -35.392;
   1:L PR[91] 10mm/sec CNT100;
   1:  PR[GP1:91,1] = PR[GP1:90,1] + 33.393;
   1:  PR[GP1:91,2] = PR[GP1:90,2] + -35.377;
   1:L PR[91] 10mm/sec CNT100;
   1:  PR[GP1:91,1] = PR[GP1:90,1] + 40.848;
   1:  PR[GP1:91,2] = PR[GP1:90,2] + -34.442;
   1:L PR[91] 10mm/sec CNT100;
   1:  PR[GP1:91,1] = PR[GP1:90,1] + 44.682;
   1:  PR[GP1:91,2] = PR[GP1:90,2] + -33.027;
   1:L PR[91] 10mm/sec CNT100;
   1:  PR[GP1:91,1] = PR[GP1:90,1] + 50.286;
   1:  PR[GP1:91,2] = PR[GP1:90,2] + -30.987;
   1:L PR[91] 10mm/sec CNT100;
   1:  PR[GP1:91,1] = PR[GP1:90,1] + 53.561;
   1:  PR[GP1:91,2] = PR[GP1:90,2] + -28.983;
   1:L PR[91] 10mm/sec CNT100;
   1:  PR[GP1:91,1] = PR[GP1:90,1] + 59.595;
   1:  PR[GP1:91,2] = PR[GP1:90,2] + -23.974;
   1:L PR[91] 10mm/sec CNT100;
   1:  PR[GP1:91,1] = PR[GP1:90,1] + 61.446;
   1:  PR[GP1:91,2] = PR[GP1:90,2] + -22.176;
   1:L PR[91] 10mm/sec CNT100;
   1:  PR[GP1:91,1] = PR[GP1:90,1] + 66.538;
   1:  PR[GP1:91,2] = PR[GP1:90,2] + -13.632;
   1:L PR[91] 10mm/sec CNT100;
   1:  PR[GP1:91,1] = PR[GP1:90,1] + 67.427;
   1:  PR[GP1:91,2] = PR[GP1:90,2] + -12.237;
   1:L PR[91] 10mm/sec CNT100;
   1:  PR[GP1:91,1] = PR[GP1:90,1] + 67.862;
   1:  PR[GP1:91,2] = PR[GP1:90,2] + -11.064;
   1:L PR[91] 10mm/sec CNT100;
   1:  PR[GP1:91,1] = PR[GP1:90,1] + 69.767;
   1:  PR[GP1:91,2] = PR[GP1:90,2] + -0.545;
   1:L PR[91] 10mm/sec CNT100;
   1:  PR[GP1:91,1] = PR[GP1:90,1] + 69.858;
   1:  PR[GP1:91,2] = PR[GP1:90,2] + 0.258;
   1:L PR[91] 10mm/sec CNT100;
   1:  PR[GP1:91,1] = PR[GP1:90,1] + 67.990;
   1:  PR[GP1:91,2] = PR[GP1:90,2] + 10.411;
   1:L PR[91] 10mm/sec CNT100;
   1:  PR[GP1:91,1] = PR[GP1:90,1] + 67.854;
   1:  PR[GP1:91,2] = PR[GP1:90,2] + 11.641;
   1:L PR[91] 10mm/sec CNT100;
   1:  PR[GP1:91,1] = PR[GP1:90,1] + 67.424;
   1:  PR[GP1:91,2] = PR[GP1:90,2] + 12.805;
   1:L PR[91] 10mm/sec CNT100;
   1:  PR[GP1:91,1] = PR[GP1:90,1] + 62.578;
   1:  PR[GP1:91,2] = PR[GP1:90,2] + 20.982;
   1:L PR[91] 10mm/sec CNT100;
   1:  PR[GP1:91,1] = PR[GP1:90,1] + 61.454;
   1:  PR[GP1:91,2] = PR[GP1:90,2] + 22.727;
   1:L PR[91] 10mm/sec CNT100;
   1:  PR[GP1:91,1] = PR[GP1:90,1] + 59.595;
   1:  PR[GP1:91,2] = PR[GP1:90,2] + 24.532;
   1:L PR[91] 10mm/sec CNT100;
   1:  PR[GP1:91,1] = PR[GP1:90,1] + 53.561;
   1:  PR[GP1:91,2] = PR[GP1:90,2] + 29.541;
   1:L PR[91] 10mm/sec CNT100;
   1:  PR[GP1:91,1] = PR[GP1:90,1] + 50.284;
   1:  PR[GP1:91,2] = PR[GP1:90,2] + 31.546;
   1:L PR[91] 10mm/sec CNT100;
   1:  PR[GP1:91,1] = PR[GP1:90,1] + 45.502;
   1:  PR[GP1:91,2] = PR[GP1:90,2] + 33.317;
   1:L PR[91] 10mm/sec CNT100;
   1:  PR[GP1:91,1] = PR[GP1:90,1] + 40.850;
   1:  PR[GP1:91,2] = PR[GP1:90,2] + 35.000;
   1:L PR[91] 10mm/sec CNT100;
   1:  PR[GP1:91,1] = PR[GP1:90,1] + 33.393;
   1:  PR[GP1:91,2] = PR[GP1:90,2] + 35.935;
   1:L PR[91] 10mm/sec CNT100;
   1:  PR[GP1:91,1] = PR[GP1:90,1] + 32.869;
   1:  PR[GP1:91,2] = PR[GP1:90,2] + 35.950;
   1:L PR[91] 10mm/sec CNT100;
   1:  PR[GP1:91,1] = PR[GP1:90,1] + 31.562;
   1:  PR[GP1:91,2] = PR[GP1:90,2] + 35.837;
   1:L PR[91] 10mm/sec CNT100;
   1:  PR[GP1:91,1] = PR[GP1:90,1] + 24.871;
   1:  PR[GP1:91,2] = PR[GP1:90,2] + 35.393;
   1:L PR[91] 10mm/sec CNT100;
   1:  PR[GP1:91,1] = PR[GP1:90,1] + 24.371;
   1:  PR[GP1:91,2] = PR[GP1:90,2] + 35.275;
   1:L PR[91] 10mm/sec CNT100;
   1:  PR[GP1:91,1] = PR[GP1:90,1] + 16.561;
   1:  PR[GP1:91,2] = PR[GP1:90,2] + 33.029;
   1:L PR[91] 10mm/sec CNT100;
   1:  PR[GP1:91,1] = PR[GP1:90,1] + 10.046;
   1:  PR[GP1:91,2] = PR[GP1:90,2] + 29.514;
   1:L PR[91] 10mm/sec CNT100;
   1:  PR[GP1:91,1] = PR[GP1:90,1] + 7.278;
   1:  PR[GP1:91,2] = PR[GP1:90,2] + 27.263;
   1:L PR[91] 10mm/sec CNT100;
   1:  PR[GP1:91,1] = PR[GP1:90,1] + 3.552;
   1:  PR[GP1:91,2] = PR[GP1:90,2] + 23.982;
   1:L PR[91] 10mm/sec CNT100;
   1:  PR[GP1:91,1] = PR[GP1:90,1] + 1.197;
   1:  PR[GP1:91,2] = PR[GP1:90,2] + 21.109;
   1:L PR[91] 10mm/sec CNT100;
   1:  PR[GP1:91,1] = PR[GP1:90,1] + 0.596;
   1:  PR[GP1:91,2] = PR[GP1:90,2] + 20.265;
   1:L PR[91] 10mm/sec CNT100;
   1:  PR[GP1:91,1] = PR[GP1:90,1] + -1.112;
   1:L PR[91] 10mm/sec CNT100;
   1:  PR[GP1:91,1] = PR[GP1:90,1] + -1.741;
   1:  PR[GP1:91,2] = PR[GP1:90,2] + 21.151;
   1:L PR[91] 10mm/sec CNT100;
   1:  PR[GP1:91,1] = PR[GP1:90,1] + -4.051;
   1:  PR[GP1:91,2] = PR[GP1:90,2] + 23.958;
   1:L PR[91] 10mm/sec CNT100;
   1:  PR[GP1:91,1] = PR[GP1:90,1] + -7.781;
   1:  PR[GP1:91,2] = PR[GP1:90,2] + 27.242;
   1:L PR[91] 10mm/sec CNT100;
   1:  PR[GP1:91,1] = PR[GP1:90,1] + -10.544;
   1:  PR[GP1:91,2] = PR[GP1:90,2] + 29.488;
   1:L PR[91] 10mm/sec CNT100;
   1:  PR[GP1:91,1] = PR[GP1:90,1] + -17.095;
   1:  PR[GP1:91,2] = PR[GP1:90,2] + 33.033;
   1:L PR[91] 10mm/sec CNT100;
   1:  PR[GP1:91,1] = PR[GP1:90,1] + -24.894;
   1:  PR[GP1:91,2] = PR[GP1:90,2] + 35.275;
   1:L PR[91] 10mm/sec CNT100;
   1:  PR[GP1:91,1] = PR[GP1:90,1] + -25.395;
   1:  PR[GP1:91,2] = PR[GP1:90,2] + 35.394;
   1:L PR[91] 10mm/sec CNT100;
   1:  PR[GP1:91,1] = PR[GP1:90,1] + -32.088;
   1:  PR[GP1:91,2] = PR[GP1:90,2] + 35.835;
   1:L PR[91] 10mm/sec CNT100;
   1:  PR[GP1:91,1] = PR[GP1:90,1] + -33.413;
   1:  PR[GP1:91,2] = PR[GP1:90,2] + 35.949;
   1:L PR[91] 10mm/sec CNT100;
   1:  PR[GP1:91,1] = PR[GP1:90,1] + -33.944;
   1:  PR[GP1:91,2] = PR[GP1:90,2] + 35.933;
   1:L PR[91] 10mm/sec CNT100;
   1:  PR[GP1:91,1] = PR[GP1:90,1] + -41.408;
   1:  PR[GP1:91,2] = PR[GP1:90,2] + 34.994;
   1:L PR[91] 10mm/sec CNT100;
   1:  PR[GP1:91,1] = PR[GP1:90,1] + -50.830;
   1:  PR[GP1:91,2] = PR[GP1:90,2] + 31.535;
   1:L PR[91] 10mm/sec CNT100;
   1:  PR[GP1:91,1] = PR[GP1:90,1] + -54.116;
   1:  PR[GP1:91,2] = PR[GP1:90,2] + 29.514;
   1:L PR[91] 10mm/sec CNT100;
   1:  PR[GP1:91,1] = PR[GP1:90,1] + -60.148;
   1:  PR[GP1:91,2] = PR[GP1:90,2] + 24.514;
   1:L PR[91] 10mm/sec CNT100;
   1:  PR[GP1:91,1] = PR[GP1:90,1] + -61.993;
   1:  PR[GP1:91,2] = PR[GP1:90,2] + 22.719;
   1:L PR[91] 10mm/sec CNT100;
   1:  PR[GP1:91,1] = PR[GP1:90,1] + -67.081;
   1:  PR[GP1:91,2] = PR[GP1:90,2] + 14.155;
   1:L PR[91] 10mm/sec CNT100;
   1:  PR[GP1:91,1] = PR[GP1:90,1] + -67.957;
   1:  PR[GP1:91,2] = PR[GP1:90,2] + 12.772;
   1:L PR[91] 10mm/sec CNT100;
   1:  PR[GP1:91,1] = PR[GP1:90,1] + -68.393;
   1:  PR[GP1:91,2] = PR[GP1:90,2] + 11.577;
   1:L PR[91] 10mm/sec CNT100;
   1:  PR[GP1:91,1] = PR[GP1:90,1] + -70.297;
   1:  PR[GP1:91,2] = PR[GP1:90,2] + 1.084;
   1:L PR[91] 10mm/sec CNT100;
   1:  PR[GP1:91,1] = PR[GP1:90,1] + -70.384;
   1:  PR[GP1:91,2] = PR[GP1:90,2] + 0.301;
   1:L PR[91] 10mm/sec CNT100;
   1:  PR[GP1:91,1] = PR[GP1:90,1] + -68.517;
   1:  PR[GP1:91,2] = PR[GP1:90,2] + -9.836;
   1:L PR[91] 10mm/sec CNT100;
   1:  PR[GP1:91,1] = PR[GP1:90,1] + -68.386;
   1:  PR[GP1:91,2] = PR[GP1:90,2] + -11.039;
   1:L PR[91] 10mm/sec CNT100;
   1:  PR[GP1:91,1] = PR[GP1:90,1] + -67.953;
   1:  PR[GP1:91,2] = PR[GP1:90,2] + -12.222;
   1:L PR[91] 10mm/sec CNT100;
   1:  PR[GP1:91,1] = PR[GP1:90,1] + -63.110;
   1:  PR[GP1:91,2] = PR[GP1:90,2] + -20.421;
   1:L PR[91] 10mm/sec CNT100;
   1:  PR[GP1:91,1] = PR[GP1:90,1] + -62.001;
   1:  PR[GP1:91,2] = PR[GP1:90,2] + -22.154;
   1:L PR[91] 10mm/sec CNT100;
   1:  PR[GP1:91,1] = PR[GP1:90,1] + -60.148;
   1:  PR[GP1:91,2] = PR[GP1:90,2] + -23.956;
   1:L PR[91] 10mm/sec CNT100;
   1:  PR[GP1:91,1] = PR[GP1:90,1] + -54.116;
   1:  PR[GP1:91,2] = PR[GP1:90,2] + -28.956;
   1:L PR[91] 10mm/sec CNT100;
   1:  PR[GP1:91,1] = PR[GP1:90,1] + -50.829;
   1:  PR[GP1:91,2] = PR[GP1:90,2] + -30.977;
   1:L PR[91] 10mm/sec CNT100;
   1:  PR[GP1:91,1] = PR[GP1:90,1] + -46.046;
   1:  PR[GP1:91,2] = PR[GP1:90,2] + -32.751;
   1:L PR[91] 10mm/sec CNT100;
   1:  PR[GP1:91,1] = PR[GP1:90,1] + -41.409;
   1:  PR[GP1:91,2] = PR[GP1:90,2] + -34.436;
   1:L PR[91] 10mm/sec CNT100;
   1:  PR[GP1:91,1] = PR[GP1:90,1] + -33.944;
   1:  PR[GP1:91,2] = PR[GP1:90,2] + -35.375;
   1:L PR[91] 10mm/sec CNT100;
   1:  PR[GP1:91,1] = PR[GP1:90,1] + -33.413;
   1:  PR[GP1:91,2] = PR[GP1:90,2] + -35.391;
   1:L PR[91] 10mm/sec CNT100;
   1:  PR[GP1:91,1] = PR[GP1:90,1] + -32.088;
   1:  PR[GP1:91,2] = PR[GP1:90,2] + -35.277;
   1:L PR[91] 10mm/sec CNT100;
   1:  PR[GP1:91,1] = PR[GP1:90,1] + -25.398;
   1:  PR[GP1:91,2] = PR[GP1:90,2] + -34.836;
   1:L PR[91] 10mm/sec CNT100;
   1:  PR[GP1:91,1] = PR[GP1:90,1] + -24.907;
   1:  PR[GP1:91,2] = PR[GP1:90,2] + -34.723;
   1:L PR[91] 10mm/sec CNT100;
   1:  PR[GP1:91,1] = PR[GP1:90,1] + -17.126;
   1:  PR[GP1:91,2] = PR[GP1:90,2] + -32.489;
   1:L PR[91] 10mm/sec CNT100;
   1:  PR[GP1:91,1] = PR[GP1:90,1] + -16.235;
   1:  PR[GP1:91,2] = PR[GP1:90,2] + -31.967;
   1:L PR[91] 10mm/sec CNT100;
   1:  PR[GP1:91,1] = PR[GP1:90,1] + -9.907;
   1:  PR[GP1:91,2] = PR[GP1:90,2] + -28.522;
   1:L PR[91] 10mm/sec CNT100;
   1:  PR[GP1:91,1] = PR[GP1:90,1] + -7.817;
   1:  PR[GP1:91,2] = PR[GP1:90,2] + -26.719;
   1:L PR[91] 10mm/sec CNT100;
   1:  PR[GP1:91,1] = PR[GP1:90,1] + -4.066;
   1:  PR[GP1:91,2] = PR[GP1:90,2] + -23.417;
   1:L PR[91] 10mm/sec CNT100;
   1:  PR[GP1:91,1] = PR[GP1:90,1] + -1.756;
   1:  PR[GP1:91,2] = PR[GP1:90,2] + -20.614;
   1:L PR[91] 10mm/sec CNT100;
   1:  PR[GP1:91,1] = PR[GP1:90,1] + -1.113;
   1:  PR[GP1:91,2] = PR[GP1:90,2] + -19.707;
   1:L PR[91] 10mm/sec CNT100;
   1:  PR[GP1:91,1] = PR[GP1:90,1] + 0.600;
   1:L PR[91] 10mm/sec CNT100;
   1:  PR[GP1:91,1] = PR[GP1:90,1] + 0.815;
   1:  PR[GP1:91,2] = PR[GP1:90,2] + -20.455;
   1:  PR[GP1:91,3] = PR[GP1:90,3] + 45.445;
   1:L PR[91] 10mm/sec CNT100;
   1:  PR[GP1:91,1] = PR[GP1:90,1] + 3.341;
   1:  PR[GP1:91,2] = PR[GP1:90,2] + -23.527;
   1:L PR[91] 10mm/sec CNT100;
   1:  PR[GP1:91,1] = PR[GP1:90,1] + 6.834;
   1:  PR[GP1:91,2] = PR[GP1:90,2] + -26.603;
   1:L PR[91] 10mm/sec CNT100;
   1:  PR[GP1:91,1] = PR[GP1:90,1] + 9.163;
   1:  PR[GP1:91,2] = PR[GP1:90,2] + -28.615;
   1:L PR[91] 10mm/sec CNT100;
   1:  PR[GP1:91,1] = PR[GP1:90,1] + 15.290;
   1:  PR[GP1:91,2] = PR[GP1:90,2] + -31.941;
   1:L PR[91] 10mm/sec CNT100;
   1:  PR[GP1:91,1] = PR[GP1:90,1] + 16.338;
   1:  PR[GP1:91,2] = PR[GP1:90,2] + -32.554;
   1:L PR[91] 10mm/sec CNT100;
   1:  PR[GP1:91,1] = PR[GP1:90,1] + 24.009;
   1:  PR[GP1:91,2] = PR[GP1:90,2] + -34.757;
   1:L PR[91] 10mm/sec CNT100;
   1:  PR[GP1:91,1] = PR[GP1:90,1] + 24.698;
   1:  PR[GP1:91,2] = PR[GP1:90,2] + -34.915;
   1:L PR[91] 10mm/sec CNT100;
   1:  PR[GP1:91,1] = PR[GP1:90,1] + 32.855;
   1:  PR[GP1:91,2] = PR[GP1:90,2] + -35.457;
   1:L PR[91] 10mm/sec CNT100;
   1:  PR[GP1:91,1] = PR[GP1:90,1] + 40.768;
   1:  PR[GP1:91,2] = PR[GP1:90,2] + -34.454;
   1:L PR[91] 10mm/sec CNT100;
   1:  PR[GP1:91,1] = PR[GP1:90,1] + 49.939;
   1:  PR[GP1:91,2] = PR[GP1:90,2] + -31.101;
   1:L PR[91] 10mm/sec CNT100;
   1:  PR[GP1:91,1] = PR[GP1:90,1] + 53.624;
   1:  PR[GP1:91,2] = PR[GP1:90,2] + -28.847;
   1:L PR[91] 10mm/sec CNT100;
   1:  PR[GP1:91,1] = PR[GP1:90,1] + 59.067;
   1:  PR[GP1:91,2] = PR[GP1:90,2] + -24.328;
   1:L PR[91] 10mm/sec CNT100;
   1:  PR[GP1:91,1] = PR[GP1:90,1] + 61.294;
   1:  PR[GP1:91,2] = PR[GP1:90,2] + -22.165;
   1:L PR[91] 10mm/sec CNT100;
   1:  PR[GP1:91,1] = PR[GP1:90,1] + 65.984;
   1:  PR[GP1:91,2] = PR[GP1:90,2] + -14.297;
   1:L PR[91] 10mm/sec CNT100;
   1:  PR[GP1:91,1] = PR[GP1:90,1] + 67.169;
   1:  PR[GP1:91,2] = PR[GP1:90,2] + -12.435;
   1:L PR[91] 10mm/sec CNT100;
   1:  PR[GP1:91,1] = PR[GP1:90,1] + 67.758;
   1:  PR[GP1:91,2] = PR[GP1:90,2] + -10.846;
   1:L PR[91] 10mm/sec CNT100;
   1:  PR[GP1:91,1] = PR[GP1:90,1] + 69.542;
   1:  PR[GP1:91,2] = PR[GP1:90,2] + -0.999;
   1:L PR[91] 10mm/sec CNT100;
   1:  PR[GP1:91,1] = PR[GP1:90,1] + 69.684;
   1:  PR[GP1:91,2] = PR[GP1:90,2] + 0.258;
   1:L PR[91] 10mm/sec CNT100;
   1:  PR[GP1:91,1] = PR[GP1:90,1] + 67.933;
   1:  PR[GP1:91,2] = PR[GP1:90,2] + 9.779;
   1:L PR[91] 10mm/sec CNT100;
   1:  PR[GP1:91,1] = PR[GP1:90,1] + 67.751;
   1:  PR[GP1:91,2] = PR[GP1:90,2] + 11.424;
   1:L PR[91] 10mm/sec CNT100;
   1:  PR[GP1:91,1] = PR[GP1:90,1] + 67.166;
   1:  PR[GP1:91,2] = PR[GP1:90,2] + 13.003;
   1:L PR[91] 10mm/sec CNT100;
   1:  PR[GP1:91,1] = PR[GP1:90,1] + 62.655;
   1:  PR[GP1:91,2] = PR[GP1:90,2] + 20.616;
   1:L PR[91] 10mm/sec CNT100;
   1:  PR[GP1:91,1] = PR[GP1:90,1] + 61.302;
   1:  PR[GP1:91,2] = PR[GP1:90,2] + 22.715;
   1:L PR[91] 10mm/sec CNT100;
   1:  PR[GP1:91,1] = PR[GP1:90,1] + 59.067;
   1:  PR[GP1:91,2] = PR[GP1:90,2] + 24.886;
   1:L PR[91] 10mm/sec CNT100;
   1:  PR[GP1:91,1] = PR[GP1:90,1] + 53.624;
   1:  PR[GP1:91,2] = PR[GP1:90,2] + 29.405;
   1:L PR[91] 10mm/sec CNT100;
   1:  PR[GP1:91,1] = PR[GP1:90,1] + 49.938;
   1:  PR[GP1:91,2] = PR[GP1:90,2] + 31.660;
   1:L PR[91] 10mm/sec CNT100;
   1:  PR[GP1:91,1] = PR[GP1:90,1] + 45.813;
   1:  PR[GP1:91,2] = PR[GP1:90,2] + 33.188;
   1:L PR[91] 10mm/sec CNT100;
   1:  PR[GP1:91,1] = PR[GP1:90,1] + 40.769;
   1:  PR[GP1:91,2] = PR[GP1:90,2] + 35.012;
   1:L PR[91] 10mm/sec CNT100;
   1:  PR[GP1:91,1] = PR[GP1:90,1] + 32.854;
   1:  PR[GP1:91,2] = PR[GP1:90,2] + 36.015;
   1:L PR[91] 10mm/sec CNT100;
   1:  PR[GP1:91,1] = PR[GP1:90,1] + 24.692;
   1:  PR[GP1:91,2] = PR[GP1:90,2] + 35.473;
   1:L PR[91] 10mm/sec CNT100;
   1:  PR[GP1:91,1] = PR[GP1:90,1] + 23.991;
   1:  PR[GP1:91,2] = PR[GP1:90,2] + 35.307;
   1:L PR[91] 10mm/sec CNT100;
   1:  PR[GP1:91,1] = PR[GP1:90,1] + 16.303;
   1:  PR[GP1:91,2] = PR[GP1:90,2] + 33.097;
   1:L PR[91] 10mm/sec CNT100;
   1:  PR[GP1:91,1] = PR[GP1:90,1] + 9.873;
   1:  PR[GP1:91,2] = PR[GP1:90,2] + 29.628;
   1:L PR[91] 10mm/sec CNT100;
   1:  PR[GP1:91,1] = PR[GP1:90,1] + 6.794;
   1:  PR[GP1:91,2] = PR[GP1:90,2] + 27.124;
   1:L PR[91] 10mm/sec CNT100;
   1:  PR[GP1:91,1] = PR[GP1:90,1] + 3.324;
   1:  PR[GP1:91,2] = PR[GP1:90,2] + 24.068;
   1:L PR[91] 10mm/sec CNT100;
   1:  PR[GP1:91,1] = PR[GP1:90,1] + 0.485;
   1:  PR[GP1:91,2] = PR[GP1:90,2] + 20.590;
   1:L PR[91] 10mm/sec CNT100;
   1:  PR[GP1:91,1] = PR[GP1:90,1] + -1.025;
   1:L PR[91] 10mm/sec CNT100;
   1:  PR[GP1:91,1] = PR[GP1:90,1] + -1.309;
   1:  PR[GP1:91,2] = PR[GP1:90,2] + 20.991;
   1:L PR[91] 10mm/sec CNT100;
   1:  PR[GP1:91,1] = PR[GP1:90,1] + -3.824;
   1:  PR[GP1:91,2] = PR[GP1:90,2] + 24.045;
   1:L PR[91] 10mm/sec CNT100;
   1:  PR[GP1:91,1] = PR[GP1:90,1] + -7.298;
   1:  PR[GP1:91,2] = PR[GP1:90,2] + 27.104;
   1:L PR[91] 10mm/sec CNT100;
   1:  PR[GP1:91,1] = PR[GP1:90,1] + -10.371;
   1:  PR[GP1:91,2] = PR[GP1:90,2] + 29.603;
   1:L PR[91] 10mm/sec CNT100;
   1:  PR[GP1:91,1] = PR[GP1:90,1] + -16.836;
   1:  PR[GP1:91,2] = PR[GP1:90,2] + 33.101;
   1:L PR[91] 10mm/sec CNT100;
   1:  PR[GP1:91,1] = PR[GP1:90,1] + -24.514;
   1:  PR[GP1:91,2] = PR[GP1:90,2] + 35.308;
   1:L PR[91] 10mm/sec CNT100;
   1:  PR[GP1:91,1] = PR[GP1:90,1] + -25.216;
   1:  PR[GP1:91,2] = PR[GP1:90,2] + 35.474;
   1:L PR[91] 10mm/sec CNT100;
   1:  PR[GP1:91,1] = PR[GP1:90,1] + -33.403;
   1:  PR[GP1:91,2] = PR[GP1:90,2] + 36.014;
   1:L PR[91] 10mm/sec CNT100;
   1:  PR[GP1:91,1] = PR[GP1:90,1] + -41.329;
   1:  PR[GP1:91,2] = PR[GP1:90,2] + 35.006;
   1:L PR[91] 10mm/sec CNT100;
   1:  PR[GP1:91,1] = PR[GP1:90,1] + -50.486;
   1:  PR[GP1:91,2] = PR[GP1:90,2] + 31.648;
   1:L PR[91] 10mm/sec CNT100;
   1:  PR[GP1:91,1] = PR[GP1:90,1] + -54.182;
   1:  PR[GP1:91,2] = PR[GP1:90,2] + 29.375;
   1:L PR[91] 10mm/sec CNT100;
   1:  PR[GP1:91,1] = PR[GP1:90,1] + -59.625;
   1:  PR[GP1:91,2] = PR[GP1:90,2] + 24.863;
   1:L PR[91] 10mm/sec CNT100;
   1:  PR[GP1:91,1] = PR[GP1:90,1] + -61.846;
   1:  PR[GP1:91,2] = PR[GP1:90,2] + 22.703;
   1:L PR[91] 10mm/sec CNT100;
   1:  PR[GP1:91,1] = PR[GP1:90,1] + -66.531;
   1:  PR[GP1:91,2] = PR[GP1:90,2] + 14.816;
   1:L PR[91] 10mm/sec CNT100;
   1:  PR[GP1:91,1] = PR[GP1:90,1] + -67.700;
   1:  PR[GP1:91,2] = PR[GP1:90,2] + 12.969;
   1:L PR[91] 10mm/sec CNT100;
   1:  PR[GP1:91,1] = PR[GP1:90,1] + -68.291;
   1:  PR[GP1:91,2] = PR[GP1:90,2] + 11.352;
   1:L PR[91] 10mm/sec CNT100;
   1:  PR[GP1:91,1] = PR[GP1:90,1] + -70.074;
   1:  PR[GP1:91,2] = PR[GP1:90,2] + 1.527;
   1:L PR[91] 10mm/sec CNT100;
   1:  PR[GP1:91,1] = PR[GP1:90,1] + -70.210;
   1:  PR[GP1:91,2] = PR[GP1:90,2] + 0.301;
   1:L PR[91] 10mm/sec CNT100;
   1:  PR[GP1:91,1] = PR[GP1:90,1] + -68.459;
   1:  PR[GP1:91,2] = PR[GP1:90,2] + -9.204;
   1:L PR[91] 10mm/sec CNT100;
   1:  PR[GP1:91,1] = PR[GP1:90,1] + -68.284;
   1:  PR[GP1:91,2] = PR[GP1:90,2] + -10.814;
   1:L PR[91] 10mm/sec CNT100;
   1:  PR[GP1:91,1] = PR[GP1:90,1] + -67.697;
   1:  PR[GP1:91,2] = PR[GP1:90,2] + -12.419;
   1:L PR[91] 10mm/sec CNT100;
   1:  PR[GP1:91,1] = PR[GP1:90,1] + -63.187;
   1:  PR[GP1:91,2] = PR[GP1:90,2] + -20.053;
   1:L PR[91] 10mm/sec CNT100;
   1:  PR[GP1:91,1] = PR[GP1:90,1] + -61.853;
   1:  PR[GP1:91,2] = PR[GP1:90,2] + -22.138;
   1:L PR[91] 10mm/sec CNT100;
   1:  PR[GP1:91,1] = PR[GP1:90,1] + -59.625;
   1:  PR[GP1:91,2] = PR[GP1:90,2] + -24.305;
   1:L PR[91] 10mm/sec CNT100;
   1:  PR[GP1:91,1] = PR[GP1:90,1] + -54.182;
   1:  PR[GP1:91,2] = PR[GP1:90,2] + -28.817;
   1:L PR[91] 10mm/sec CNT100;
   1:  PR[GP1:91,1] = PR[GP1:90,1] + -50.485;
   1:  PR[GP1:91,2] = PR[GP1:90,2] + -31.091;
   1:L PR[91] 10mm/sec CNT100;
   1:  PR[GP1:91,1] = PR[GP1:90,1] + -46.356;
   1:  PR[GP1:91,2] = PR[GP1:90,2] + -32.621;
   1:L PR[91] 10mm/sec CNT100;
   1:  PR[GP1:91,1] = PR[GP1:90,1] + -41.330;
   1:  PR[GP1:91,2] = PR[GP1:90,2] + -34.448;
   1:L PR[91] 10mm/sec CNT100;
   1:  PR[GP1:91,1] = PR[GP1:90,1] + -33.403;
   1:  PR[GP1:91,2] = PR[GP1:90,2] + -35.456;
   1:L PR[91] 10mm/sec CNT100;
   1:  PR[GP1:91,1] = PR[GP1:90,1] + -25.222;
   1:  PR[GP1:91,2] = PR[GP1:90,2] + -34.916;
   1:L PR[91] 10mm/sec CNT100;
   1:  PR[GP1:91,1] = PR[GP1:90,1] + -24.532;
   1:  PR[GP1:91,2] = PR[GP1:90,2] + -34.758;
   1:L PR[91] 10mm/sec CNT100;
   1:  PR[GP1:91,1] = PR[GP1:90,1] + -16.871;
   1:  PR[GP1:91,2] = PR[GP1:90,2] + -32.558;
   1:L PR[91] 10mm/sec CNT100;
   1:  PR[GP1:91,1] = PR[GP1:90,1] + -15.825;
   1:  PR[GP1:91,2] = PR[GP1:90,2] + -31.945;
   1:L PR[91] 10mm/sec CNT100;
   1:  PR[GP1:91,1] = PR[GP1:90,1] + -9.664;
   1:  PR[GP1:91,2] = PR[GP1:90,2] + -28.591;
   1:L PR[91] 10mm/sec CNT100;
   1:  PR[GP1:91,1] = PR[GP1:90,1] + -7.337;
   1:  PR[GP1:91,2] = PR[GP1:90,2] + -26.584;
   1:L PR[91] 10mm/sec CNT100;
   1:  PR[GP1:91,1] = PR[GP1:90,1] + -3.840;
   1:  PR[GP1:91,2] = PR[GP1:90,2] + -23.505;
   1:L PR[91] 10mm/sec CNT100;
   1:  PR[GP1:91,1] = PR[GP1:90,1] + -1.326;
   1:  PR[GP1:91,2] = PR[GP1:90,2] + -20.454;
   1:L PR[91] 10mm/sec CNT100;
   1:  PR[GP1:91,1] = PR[GP1:90,1] + -1.026;
   1:  PR[GP1:91,2] = PR[GP1:90,2] + -20.032;
   1:L PR[91] 10mm/sec CNT100;
   1:  PR[GP1:91,1] = PR[GP1:90,1] + 0.514;
   1:L PR[91] 10mm/sec CNT100;
   1:  PR[GP1:91,1] = PR[GP1:90,1] + 3.114;
   1:  PR[GP1:91,2] = PR[GP1:90,2] + -23.614;
   1:  PR[GP1:91,3] = PR[GP1:90,3] + 46.055;
   1:L PR[91] 10mm/sec CNT100;
   1:  PR[GP1:91,1] = PR[GP1:90,1] + 6.352;
   1:  PR[GP1:91,2] = PR[GP1:90,2] + -26.466;
   1:L PR[91] 10mm/sec CNT100;
   1:  PR[GP1:91,1] = PR[GP1:90,1] + 8.918;
   1:  PR[GP1:91,2] = PR[GP1:90,2] + -28.684;
   1:L PR[91] 10mm/sec CNT100;
   1:  PR[GP1:91,1] = PR[GP1:90,1] + 14.879;
   1:  PR[GP1:91,2] = PR[GP1:90,2] + -31.919;
   1:L PR[91] 10mm/sec CNT100;
   1:  PR[GP1:91,1] = PR[GP1:90,1] + 16.083;
   1:  PR[GP1:91,2] = PR[GP1:90,2] + -32.624;
   1:L PR[91] 10mm/sec CNT100;
   1:  PR[GP1:91,1] = PR[GP1:90,1] + 23.633;
   1:  PR[GP1:91,2] = PR[GP1:90,2] + -34.792;
   1:L PR[91] 10mm/sec CNT100;
   1:  PR[GP1:91,1] = PR[GP1:90,1] + 24.521;
   1:  PR[GP1:91,2] = PR[GP1:90,2] + -34.995;
   1:L PR[91] 10mm/sec CNT100;
   1:  PR[GP1:91,1] = PR[GP1:90,1] + 32.552;
   1:  PR[GP1:91,2] = PR[GP1:90,2] + -35.529;
   1:L PR[91] 10mm/sec CNT100;
   1:  PR[GP1:91,1] = PR[GP1:90,1] + 35.912;
   1:  PR[GP1:91,2] = PR[GP1:90,2] + -35.065;
   1:L PR[91] 10mm/sec CNT100;
   1:  PR[GP1:91,1] = PR[GP1:90,1] + 40.688;
   1:  PR[GP1:91,2] = PR[GP1:90,2] + -34.467;
   1:L PR[91] 10mm/sec CNT100;
   1:  PR[GP1:91,1] = PR[GP1:90,1] + 49.594;
   1:  PR[GP1:91,2] = PR[GP1:90,2] + -31.215;
   1:L PR[91] 10mm/sec CNT100;
   1:  PR[GP1:91,1] = PR[GP1:90,1] + 53.687;
   1:  PR[GP1:91,2] = PR[GP1:90,2] + -28.711;
   1:L PR[91] 10mm/sec CNT100;
   1:  PR[GP1:91,1] = PR[GP1:90,1] + 58.539;
   1:  PR[GP1:91,2] = PR[GP1:90,2] + -24.683;
   1:L PR[91] 10mm/sec CNT100;
   1:  PR[GP1:91,1] = PR[GP1:90,1] + 61.142;
   1:  PR[GP1:91,2] = PR[GP1:90,2] + -22.154;
   1:L PR[91] 10mm/sec CNT100;
   1:  PR[GP1:91,1] = PR[GP1:90,1] + 65.429;
   1:  PR[GP1:91,2] = PR[GP1:90,2] + -14.962;
   1:L PR[91] 10mm/sec CNT100;
   1:  PR[GP1:91,1] = PR[GP1:90,1] + 66.912;
   1:  PR[GP1:91,2] = PR[GP1:90,2] + -12.633;
   1:L PR[91] 10mm/sec CNT100;
   1:  PR[GP1:91,1] = PR[GP1:90,1] + 67.654;
   1:  PR[GP1:91,2] = PR[GP1:90,2] + -10.628;
   1:L PR[91] 10mm/sec CNT100;
   1:  PR[GP1:91,1] = PR[GP1:90,1] + 69.317;
   1:  PR[GP1:91,2] = PR[GP1:90,2] + -1.452;
   1:L PR[91] 10mm/sec CNT100;
   1:  PR[GP1:91,1] = PR[GP1:90,1] + 69.510;
   1:  PR[GP1:91,2] = PR[GP1:90,2] + 0.258;
   1:L PR[91] 10mm/sec CNT100;
   1:  PR[GP1:91,1] = PR[GP1:90,1] + 67.875;
   1:  PR[GP1:91,2] = PR[GP1:90,2] + 9.146;
   1:L PR[91] 10mm/sec CNT100;
   1:  PR[GP1:91,1] = PR[GP1:90,1] + 67.647;
   1:  PR[GP1:91,2] = PR[GP1:90,2] + 11.206;
   1:L PR[91] 10mm/sec CNT100;
   1:  PR[GP1:91,1] = PR[GP1:90,1] + 66.909;
   1:  PR[GP1:91,2] = PR[GP1:90,2] + 13.201;
   1:L PR[91] 10mm/sec CNT100;
   1:  PR[GP1:91,1] = PR[GP1:90,1] + 62.731;
   1:  PR[GP1:91,2] = PR[GP1:90,2] + 20.251;
   1:L PR[91] 10mm/sec CNT100;
   1:  PR[GP1:91,1] = PR[GP1:90,1] + 61.150;
   1:  PR[GP1:91,2] = PR[GP1:90,2] + 22.704;
   1:L PR[91] 10mm/sec CNT100;
   1:  PR[GP1:91,1] = PR[GP1:90,1] + 58.539;
   1:  PR[GP1:91,2] = PR[GP1:90,2] + 25.241;
   1:L PR[91] 10mm/sec CNT100;
   1:  PR[GP1:91,1] = PR[GP1:90,1] + 53.687;
   1:  PR[GP1:91,2] = PR[GP1:90,2] + 29.269;
   1:L PR[91] 10mm/sec CNT100;
   1:  PR[GP1:91,1] = PR[GP1:90,1] + 49.592;
   1:  PR[GP1:91,2] = PR[GP1:90,2] + 31.774;
   1:L PR[91] 10mm/sec CNT100;
   1:  PR[GP1:91,1] = PR[GP1:90,1] + 46.123;
   1:  PR[GP1:91,2] = PR[GP1:90,2] + 33.058;
   1:L PR[91] 10mm/sec CNT100;
   1:  PR[GP1:91,1] = PR[GP1:90,1] + 40.689;
   1:  PR[GP1:91,2] = PR[GP1:90,2] + 35.024;
   1:L PR[91] 10mm/sec CNT100;
   1:  PR[GP1:91,1] = PR[GP1:90,1] + 35.911;
   1:  PR[GP1:91,2] = PR[GP1:90,2] + 35.623;
   1:L PR[91] 10mm/sec CNT100;
   1:  PR[GP1:91,1] = PR[GP1:90,1] + 32.773;
   1:  PR[GP1:91,2] = PR[GP1:90,2] + 36.068;
   1:L PR[91] 10mm/sec CNT100;
   1:  PR[GP1:91,1] = PR[GP1:90,1] + 32.562;
   1:  PR[GP1:91,2] = PR[GP1:90,2] + 36.088;
   1:L PR[91] 10mm/sec CNT100;
   1:  PR[GP1:91,1] = PR[GP1:90,1] + 24.513;
   1:  PR[GP1:91,2] = PR[GP1:90,2] + 35.553;
   1:L PR[91] 10mm/sec CNT100;
   1:  PR[GP1:91,1] = PR[GP1:90,1] + 23.610;
   1:  PR[GP1:91,2] = PR[GP1:90,2] + 35.340;
   1:L PR[91] 10mm/sec CNT100;
   1:  PR[GP1:91,1] = PR[GP1:90,1] + 16.045;
   1:  PR[GP1:91,2] = PR[GP1:90,2] + 33.165;
   1:L PR[91] 10mm/sec CNT100;
   1:  PR[GP1:91,1] = PR[GP1:90,1] + 9.700;
   1:  PR[GP1:91,2] = PR[GP1:90,2] + 29.742;
   1:L PR[91] 10mm/sec CNT100;
   1:  PR[GP1:91,1] = PR[GP1:90,1] + 6.309;
   1:  PR[GP1:91,2] = PR[GP1:90,2] + 26.984;
   1:L PR[91] 10mm/sec CNT100;
   1:  PR[GP1:91,1] = PR[GP1:90,1] + 3.094;
   1:  PR[GP1:91,2] = PR[GP1:90,2] + 24.153;
   1:L PR[91] 10mm/sec CNT100;
   1:  PR[GP1:91,1] = PR[GP1:90,1] + 0.439;
   1:  PR[GP1:91,2] = PR[GP1:90,2] + 20.915;
   1:L PR[91] 10mm/sec CNT100;
   1:  PR[GP1:91,1] = PR[GP1:90,1] + -0.948;
   1:L PR[91] 10mm/sec CNT100;
   1:  PR[GP1:91,1] = PR[GP1:90,1] + -3.596;
   1:  PR[GP1:91,2] = PR[GP1:90,2] + 24.132;
   1:L PR[91] 10mm/sec CNT100;
   1:  PR[GP1:91,1] = PR[GP1:90,1] + -6.815;
   1:  PR[GP1:91,2] = PR[GP1:90,2] + 26.966;
   1:L PR[91] 10mm/sec CNT100;
   1:  PR[GP1:91,1] = PR[GP1:90,1] + -10.199;
   1:  PR[GP1:91,2] = PR[GP1:90,2] + 29.717;
   1:L PR[91] 10mm/sec CNT100;
   1:  PR[GP1:91,1] = PR[GP1:90,1] + -16.578;
   1:  PR[GP1:91,2] = PR[GP1:90,2] + 33.168;
   1:L PR[91] 10mm/sec CNT100;
   1:  PR[GP1:91,1] = PR[GP1:90,1] + -24.133;
   1:  PR[GP1:91,2] = PR[GP1:90,2] + 35.340;
   1:L PR[91] 10mm/sec CNT100;
   1:  PR[GP1:91,1] = PR[GP1:90,1] + -25.037;
   1:  PR[GP1:91,2] = PR[GP1:90,2] + 35.554;
   1:L PR[91] 10mm/sec CNT100;
   1:  PR[GP1:91,1] = PR[GP1:90,1] + -33.097;
   1:  PR[GP1:91,2] = PR[GP1:90,2] + 36.085;
   1:L PR[91] 10mm/sec CNT100;
   1:  PR[GP1:91,1] = PR[GP1:90,1] + -36.438;
   1:  PR[GP1:91,2] = PR[GP1:90,2] + 35.623;
   1:L PR[91] 10mm/sec CNT100;
   1:  PR[GP1:91,1] = PR[GP1:90,1] + -41.251;
   1:  PR[GP1:91,2] = PR[GP1:90,2] + 35.017;
   1:L PR[91] 10mm/sec CNT100;
   1:  PR[GP1:91,1] = PR[GP1:90,1] + -50.142;
   1:  PR[GP1:91,2] = PR[GP1:90,2] + 31.761;
   1:L PR[91] 10mm/sec CNT100;
   1:  PR[GP1:91,1] = PR[GP1:90,1] + -54.248;
   1:  PR[GP1:91,2] = PR[GP1:90,2] + 29.236;
   1:L PR[91] 10mm/sec CNT100;
   1:  PR[GP1:91,1] = PR[GP1:90,1] + -59.102;
   1:  PR[GP1:91,2] = PR[GP1:90,2] + 25.213;
   1:L PR[91] 10mm/sec CNT100;
   1:  PR[GP1:91,1] = PR[GP1:90,1] + -61.698;
   1:  PR[GP1:91,2] = PR[GP1:90,2] + 22.687;
   1:L PR[91] 10mm/sec CNT100;
   1:  PR[GP1:91,1] = PR[GP1:90,1] + -65.982;
   1:  PR[GP1:91,2] = PR[GP1:90,2] + 15.476;
   1:L PR[91] 10mm/sec CNT100;
   1:  PR[GP1:91,1] = PR[GP1:90,1] + -67.444;
   1:  PR[GP1:91,2] = PR[GP1:90,2] + 13.165;
   1:L PR[91] 10mm/sec CNT100;
   1:  PR[GP1:91,1] = PR[GP1:90,1] + -68.189;
   1:  PR[GP1:91,2] = PR[GP1:90,2] + 11.126;
   1:L PR[91] 10mm/sec CNT100;
   1:  PR[GP1:91,1] = PR[GP1:90,1] + -69.851;
   1:  PR[GP1:91,2] = PR[GP1:90,2] + 1.971;
   1:L PR[91] 10mm/sec CNT100;
   1:  PR[GP1:91,1] = PR[GP1:90,1] + -70.036;
   1:  PR[GP1:91,2] = PR[GP1:90,2] + 0.301;
   1:L PR[91] 10mm/sec CNT100;
   1:  PR[GP1:91,1] = PR[GP1:90,1] + -68.402;
   1:  PR[GP1:91,2] = PR[GP1:90,2] + -8.572;
   1:L PR[91] 10mm/sec CNT100;
   1:  PR[GP1:91,1] = PR[GP1:90,1] + -68.182;
   1:  PR[GP1:91,2] = PR[GP1:90,2] + -10.589;
   1:L PR[91] 10mm/sec CNT100;
   1:  PR[GP1:91,1] = PR[GP1:90,1] + -67.441;
   1:  PR[GP1:91,2] = PR[GP1:90,2] + -12.616;
   1:L PR[91] 10mm/sec CNT100;
   1:  PR[GP1:91,1] = PR[GP1:90,1] + -63.265;
   1:  PR[GP1:91,2] = PR[GP1:90,2] + -19.685;
   1:L PR[91] 10mm/sec CNT100;
   1:  PR[GP1:91,1] = PR[GP1:90,1] + -61.705;
   1:  PR[GP1:91,2] = PR[GP1:90,2] + -22.122;
   1:L PR[91] 10mm/sec CNT100;
   1:  PR[GP1:91,1] = PR[GP1:90,1] + -59.102;
   1:  PR[GP1:91,2] = PR[GP1:90,2] + -24.654;
   1:L PR[91] 10mm/sec CNT100;
   1:  PR[GP1:91,1] = PR[GP1:90,1] + -54.248;
   1:  PR[GP1:91,2] = PR[GP1:90,2] + -28.678;
   1:L PR[91] 10mm/sec CNT100;
   1:  PR[GP1:91,1] = PR[GP1:90,1] + -50.141;
   1:  PR[GP1:91,2] = PR[GP1:90,2] + -31.204;
   1:L PR[91] 10mm/sec CNT100;
   1:  PR[GP1:91,1] = PR[GP1:90,1] + -46.670;
   1:  PR[GP1:91,2] = PR[GP1:90,2] + -32.490;
   1:L PR[91] 10mm/sec CNT100;
   1:  PR[GP1:91,1] = PR[GP1:90,1] + -41.252;
   1:  PR[GP1:91,2] = PR[GP1:90,2] + -34.459;
   1:L PR[91] 10mm/sec CNT100;
   1:  PR[GP1:91,1] = PR[GP1:90,1] + -36.437;
   1:  PR[GP1:91,2] = PR[GP1:90,2] + -35.065;
   1:L PR[91] 10mm/sec CNT100;
   1:  PR[GP1:91,1] = PR[GP1:90,1] + -33.321;
   1:  PR[GP1:91,2] = PR[GP1:90,2] + -35.508;
   1:L PR[91] 10mm/sec CNT100;
   1:  PR[GP1:91,1] = PR[GP1:90,1] + -33.112;
   1:  PR[GP1:91,2] = PR[GP1:90,2] + -35.528;
   1:L PR[91] 10mm/sec CNT100;
   1:  PR[GP1:91,1] = PR[GP1:90,1] + -25.045;
   1:  PR[GP1:91,2] = PR[GP1:90,2] + -34.996;
   1:L PR[91] 10mm/sec CNT100;
   1:  PR[GP1:91,1] = PR[GP1:90,1] + -24.157;
   1:  PR[GP1:91,2] = PR[GP1:90,2] + -34.793;
   1:L PR[91] 10mm/sec CNT100;
   1:  PR[GP1:91,1] = PR[GP1:90,1] + -16.617;
   1:  PR[GP1:91,2] = PR[GP1:90,2] + -32.627;
   1:L PR[91] 10mm/sec CNT100;
   1:  PR[GP1:91,1] = PR[GP1:90,1] + -15.414;
   1:  PR[GP1:91,2] = PR[GP1:90,2] + -31.923;
   1:L PR[91] 10mm/sec CNT100;
   1:  PR[GP1:91,1] = PR[GP1:90,1] + -9.420;
   1:  PR[GP1:91,2] = PR[GP1:90,2] + -28.660;
   1:L PR[91] 10mm/sec CNT100;
   1:  PR[GP1:91,1] = PR[GP1:90,1] + -6.857;
   1:  PR[GP1:91,2] = PR[GP1:90,2] + -26.449;
   1:L PR[91] 10mm/sec CNT100;
   1:  PR[GP1:91,1] = PR[GP1:90,1] + -3.614;
   1:  PR[GP1:91,2] = PR[GP1:90,2] + -23.594;
   1:L PR[91] 10mm/sec CNT100;
   1:  PR[GP1:91,1] = PR[GP1:90,1] + -0.947;
   1:  PR[GP1:91,2] = PR[GP1:90,2] + -20.357;
   1:L PR[91] 10mm/sec CNT100;
   1:  PR[GP1:91,1] = PR[GP1:90,1] + 0.435;
   1:L PR[91] 10mm/sec CNT100;
   1:  PR[GP1:91,1] = PR[GP1:90,1] + 2.886;
   1:  PR[GP1:91,2] = PR[GP1:90,2] + -23.701;
   1:  PR[GP1:91,3] = PR[GP1:90,3] + 46.665;
   1:L PR[91] 10mm/sec CNT100;
   1:  PR[GP1:91,1] = PR[GP1:90,1] + 5.871;
   1:  PR[GP1:91,2] = PR[GP1:90,2] + -26.330;
   1:L PR[91] 10mm/sec CNT100;
   1:  PR[GP1:91,1] = PR[GP1:90,1] + 8.674;
   1:  PR[GP1:91,2] = PR[GP1:90,2] + -28.752;
   1:L PR[91] 10mm/sec CNT100;
   1:  PR[GP1:91,1] = PR[GP1:90,1] + 14.469;
   1:  PR[GP1:91,2] = PR[GP1:90,2] + -31.897;
   1:L PR[91] 10mm/sec CNT100;
   1:  PR[GP1:91,1] = PR[GP1:90,1] + 15.829;
   1:  PR[GP1:91,2] = PR[GP1:90,2] + -32.693;
   1:L PR[91] 10mm/sec CNT100;
   1:  PR[GP1:91,1] = PR[GP1:90,1] + 23.258;
   1:  PR[GP1:91,2] = PR[GP1:90,2] + -34.827;
   1:L PR[91] 10mm/sec CNT100;
   1:  PR[GP1:91,1] = PR[GP1:90,1] + 24.345;
   1:  PR[GP1:91,2] = PR[GP1:90,2] + -35.076;
   1:L PR[91] 10mm/sec CNT100;
   1:  PR[GP1:91,1] = PR[GP1:90,1] + 32.252;
   1:  PR[GP1:91,2] = PR[GP1:90,2] + -35.601;
   1:L PR[91] 10mm/sec CNT100;
   1:  PR[GP1:91,1] = PR[GP1:90,1] + 38.149;
   1:  PR[GP1:91,2] = PR[GP1:90,2] + -34.787;
   1:L PR[91] 10mm/sec CNT100;
   1:  PR[GP1:91,1] = PR[GP1:90,1] + 40.607;
   1:  PR[GP1:91,2] = PR[GP1:90,2] + -34.479;
   1:L PR[91] 10mm/sec CNT100;
   1:  PR[GP1:91,1] = PR[GP1:90,1] + 49.248;
   1:  PR[GP1:91,2] = PR[GP1:90,2] + -31.329;
   1:L PR[91] 10mm/sec CNT100;
   1:  PR[GP1:91,1] = PR[GP1:90,1] + 53.750;
   1:  PR[GP1:91,2] = PR[GP1:90,2] + -28.575;
   1:L PR[91] 10mm/sec CNT100;
   1:  PR[GP1:91,1] = PR[GP1:90,1] + 58.011;
   1:  PR[GP1:91,2] = PR[GP1:90,2] + -25.037;
   1:L PR[91] 10mm/sec CNT100;
   1:  PR[GP1:91,1] = PR[GP1:90,1] + 60.991;
   1:  PR[GP1:91,2] = PR[GP1:90,2] + -22.142;
   1:L PR[91] 10mm/sec CNT100;
   1:  PR[GP1:91,1] = PR[GP1:90,1] + 64.874;
   1:  PR[GP1:91,2] = PR[GP1:90,2] + -15.627;
   1:L PR[91] 10mm/sec CNT100;
   1:  PR[GP1:91,1] = PR[GP1:90,1] + 66.655;
   1:  PR[GP1:91,2] = PR[GP1:90,2] + -12.831;
   1:L PR[91] 10mm/sec CNT100;
   1:  PR[GP1:91,1] = PR[GP1:90,1] + 67.551;
   1:  PR[GP1:91,2] = PR[GP1:90,2] + -10.411;
   1:L PR[91] 10mm/sec CNT100;
   1:  PR[GP1:91,1] = PR[GP1:90,1] + 69.092;
   1:  PR[GP1:91,2] = PR[GP1:90,2] + -1.906;
   1:L PR[91] 10mm/sec CNT100;
   1:  PR[GP1:91,1] = PR[GP1:90,1] + 69.336;
   1:  PR[GP1:91,2] = PR[GP1:90,2] + 0.258;
   1:L PR[91] 10mm/sec CNT100;
   1:  PR[GP1:91,1] = PR[GP1:90,1] + 67.818;
   1:  PR[GP1:91,2] = PR[GP1:90,2] + 8.513;
   1:L PR[91] 10mm/sec CNT100;
